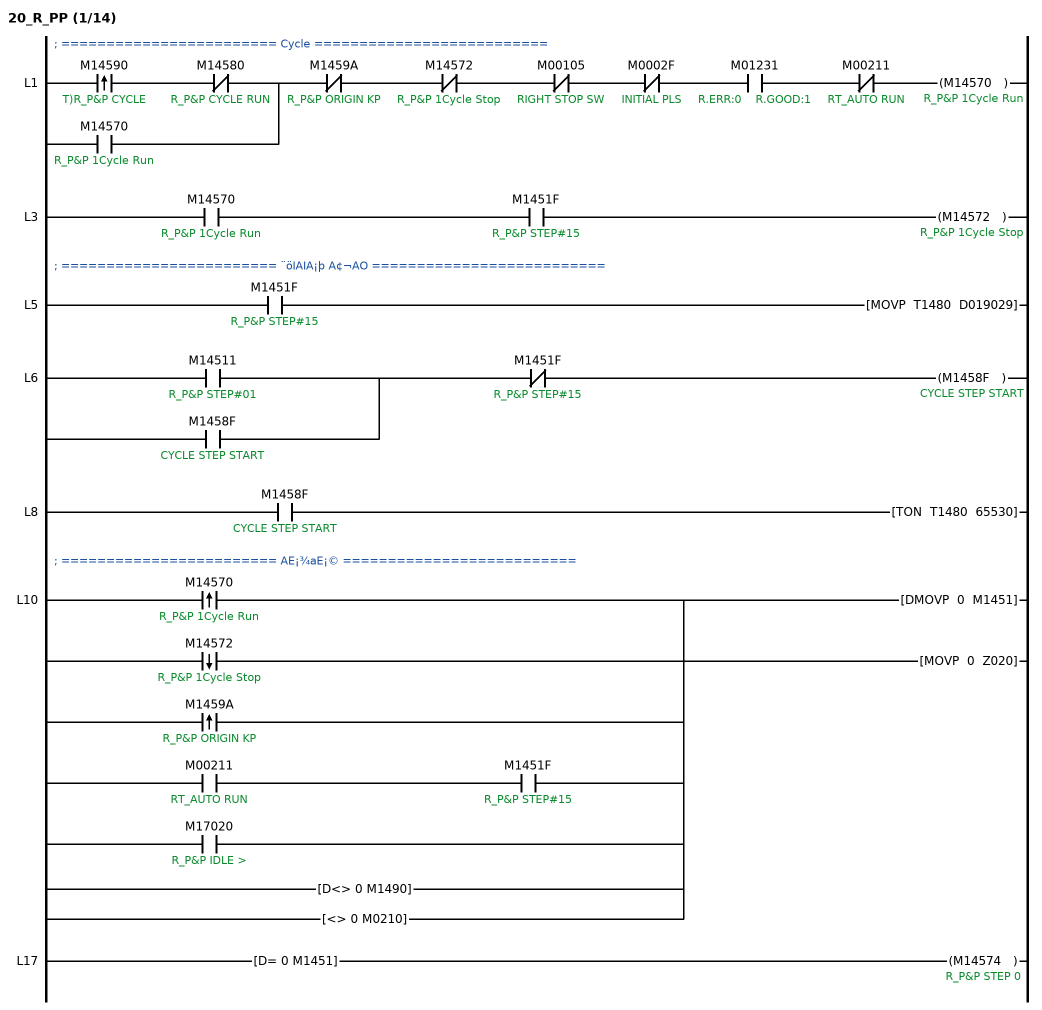
[picture p192: 20_R_PP rungs L1-L17]
// ======================== Cycle ==========================
; L1
LOADP     M14590	// T)R_P&P CYCLE
AND NOT   M14580	// R_P&P CYCLE RUN
OR        M14570	// R_P&P 1Cycle Run
AND NOT   M1459A	// R_P&P ORIGIN KP
AND NOT   M14572	// R_P&P 1Cycle Stop
AND NOT   M00105	// RIGHT STOP SW
AND NOT   M0002F	// INITIAL PLS
AND       M01231	// R.ERR:0    R.GOOD:1
AND NOT   M00211	// RT_AUTO RUN
OUT       M14570	// R_P&P 1Cycle Run
; L3
LOAD      M14570	// R_P&P 1Cycle Run
AND       M1451F	// R_P&P STEP#15
OUT       M14572	// R_P&P 1Cycle Stop
// ======================== ¨öIAIA¡þ A¢¬AO ==========================
; L5
LOAD      M1451F	// R_P&P STEP#15
MOVP      T1480 D019029
; L6
LOAD      M14511	// R_P&P STEP#01
OR        M1458F	// CYCLE STEP START
AND NOT   M1451F	// R_P&P STEP#15
OUT       M1458F	// CYCLE STEP START
; L8
LOAD      M1458F	// CYCLE STEP START
TON       T1480 65530
// ======================== AE¡¾aE¡© ==========================
; L10
LOADP     M14570	// R_P&P 1Cycle Run
ORN       M14572	// R_P&P 1Cycle Stop
ORP       M1459A	// R_P&P ORIGIN KP
LOAD      M00211	// RT_AUTO RUN
AND       M1451F	// R_P&P STEP#15
OR LOAD
OR        M17020	// R_P&P IDLE >
ORD<>     0 M1490
OR<>      0 M0210
DMOVP     0 M1451
MOVP      0 Z020
; L17
LOADD=    0 M1451
OUT       M14574	// R_P&P STEP 0

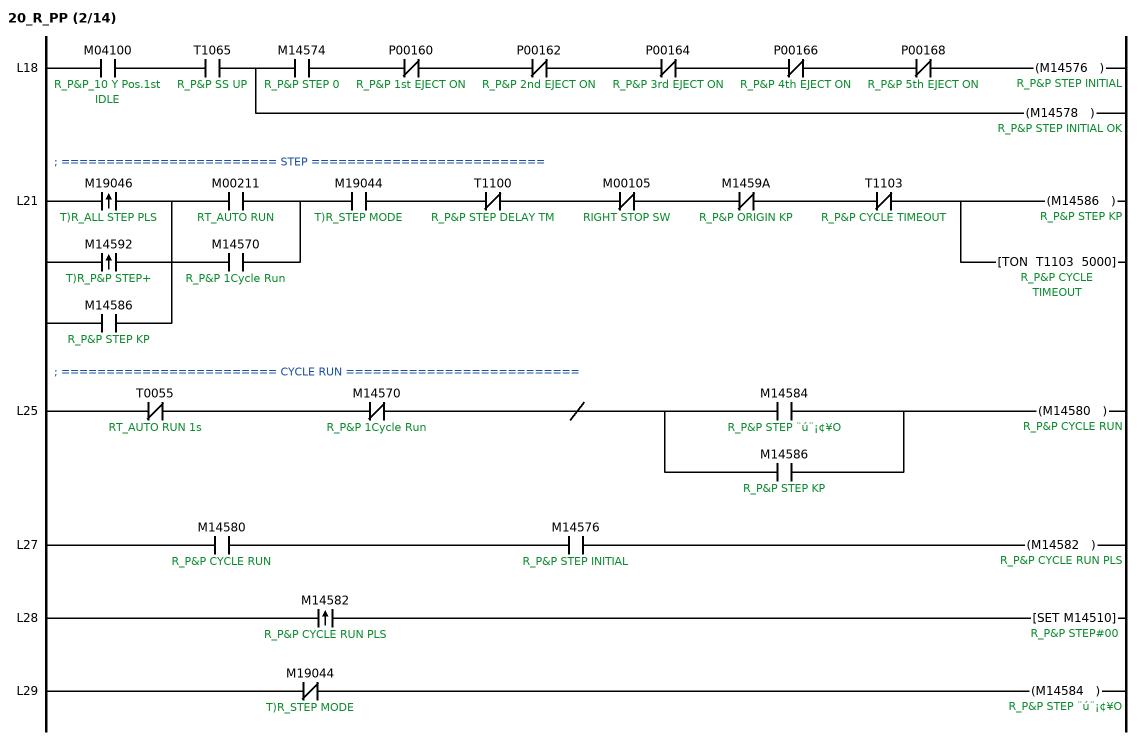
; L18
LOAD      M04100	// R_P&P_10 Y Pos.1st IDLE
AND       T1065	// R_P&P SS UP
MPUSH
AND       M14574	// R_P&P STEP 0
AND NOT   P00160	// R_P&P 1st EJECT ON
AND NOT   P00162	// R_P&P 2nd EJECT ON
AND NOT   P00164	// R_P&P 3rd EJECT ON
AND NOT   P00166	// R_P&P 4th EJECT ON
AND NOT   P00168	// R_P&P 5th EJECT ON
OUT       M14576	// R_P&P STEP INITIAL
MPOP
OUT       M14578	// R_P&P STEP INITIAL OK
// ======================== STEP ==========================
; L21
LOADP     M19046	// T)R_ALL STEP PLS
ORP       M14592	// T)R_P&P STEP+
OR        M14586	// R_P&P STEP KP
LOAD      M00211	// RT_AUTO RUN
OR        M14570	// R_P&P 1Cycle Run
AND LOAD
AND       M19044	// T)R_STEP MODE
AND NOT   T1100	// R_P&P STEP DELAY TM
AND NOT   M00105	// RIGHT STOP SW
AND NOT   M1459A	// R_P&P ORIGIN KP
AND NOT   T1103	// R_P&P CYCLE TIMEOUT
OUT       M14586	// R_P&P STEP KP
TON       T1103 5000	// R_P&P CYCLE TIMEOUT
// ======================== CYCLE RUN ==========================
; L25
LOAD NOT  T0055	// RT_AUTO RUN 1s
AND NOT   M14570	// R_P&P 1Cycle Run
NOT
LOAD      M14584	// R_P&P STEP ¨ú¨¡¢¥O
OR        M14586	// R_P&P STEP KP
AND LOAD
OUT       M14580	// R_P&P CYCLE RUN
; L27
LOAD      M14580	// R_P&P CYCLE RUN
AND       M14576	// R_P&P STEP INITIAL
OUT       M14582	// R_P&P CYCLE RUN PLS
; L28
LOADP     M14582	// R_P&P CYCLE RUN PLS
SET       M14510	// R_P&P STEP#00
; L29
LOAD NOT  M19044	// T)R_STEP MODE
OUT       M14584	// R_P&P STEP ¨ú¨¡¢¥O

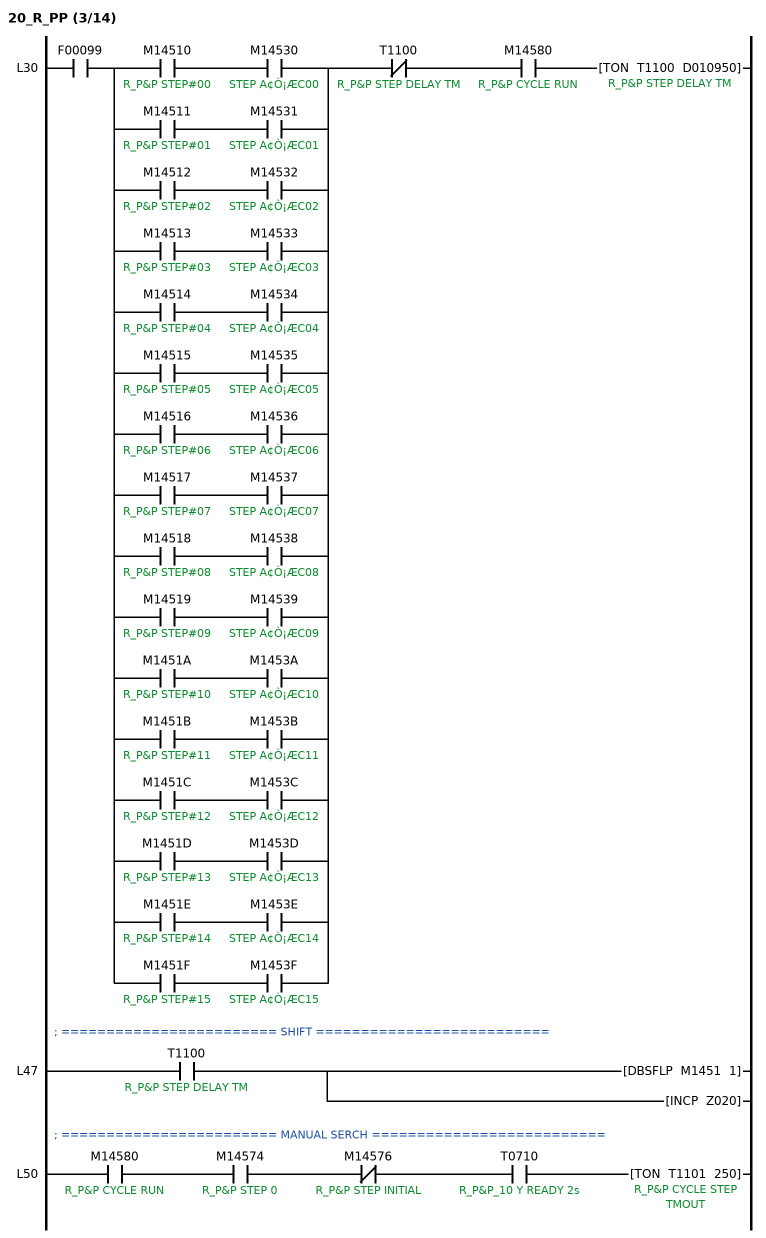
; L30
LOAD      F00099
LOAD      M14510	// R_P&P STEP#00
AND       M14530	// STEP A¢Ò¡ÆC00
LOAD      M14511	// R_P&P STEP#01
AND       M14531	// STEP A¢Ò¡ÆC01
OR LOAD
LOAD      M14512	// R_P&P STEP#02
AND       M14532	// STEP A¢Ò¡ÆC02
OR LOAD
LOAD      M14513	// R_P&P STEP#03
AND       M14533	// STEP A¢Ò¡ÆC03
OR LOAD
LOAD      M14514	// R_P&P STEP#04
AND       M14534	// STEP A¢Ò¡ÆC04
OR LOAD
LOAD      M14515	// R_P&P STEP#05
AND       M14535	// STEP A¢Ò¡ÆC05
OR LOAD
LOAD      M14516	// R_P&P STEP#06
AND       M14536	// STEP A¢Ò¡ÆC06
OR LOAD
LOAD      M14517	// R_P&P STEP#07
AND       M14537	// STEP A¢Ò¡ÆC07
OR LOAD
LOAD      M14518	// R_P&P STEP#08
AND       M14538	// STEP A¢Ò¡ÆC08
OR LOAD
LOAD      M14519	// R_P&P STEP#09
AND       M14539	// STEP A¢Ò¡ÆC09
OR LOAD
LOAD      M1451A	// R_P&P STEP#10
AND       M1453A	// STEP A¢Ò¡ÆC10
OR LOAD
LOAD      M1451B	// R_P&P STEP#11
AND       M1453B	// STEP A¢Ò¡ÆC11
OR LOAD
LOAD      M1451C	// R_P&P STEP#12
AND       M1453C	// STEP A¢Ò¡ÆC12
OR LOAD
LOAD      M1451D	// R_P&P STEP#13
AND       M1453D	// STEP A¢Ò¡ÆC13
OR LOAD
LOAD      M1451E	// R_P&P STEP#14
AND       M1453E	// STEP A¢Ò¡ÆC14
OR LOAD
LOAD      M1451F	// R_P&P STEP#15
AND       M1453F	// STEP A¢Ò¡ÆC15
OR LOAD
AND LOAD
AND NOT   T1100	// R_P&P STEP DELAY TM
AND       M14580	// R_P&P CYCLE RUN
TON       T1100 D010950	// R_P&P STEP DELAY TM
// ======================== SHIFT ==========================
; L47
LOAD      T1100	// R_P&P STEP DELAY TM
DBSFLP    M1451 1
INCP      Z020
// ======================== MANUAL SERCH ==========================
; L50
LOAD      M14580	// R_P&P CYCLE RUN
AND       M14574	// R_P&P STEP 0
AND NOT   M14576	// R_P&P STEP INITIAL
AND       T0710	// R_P&P_10 Y READY 2s
TON       T1101 250	// R_P&P CYCLE STEP TMOUT

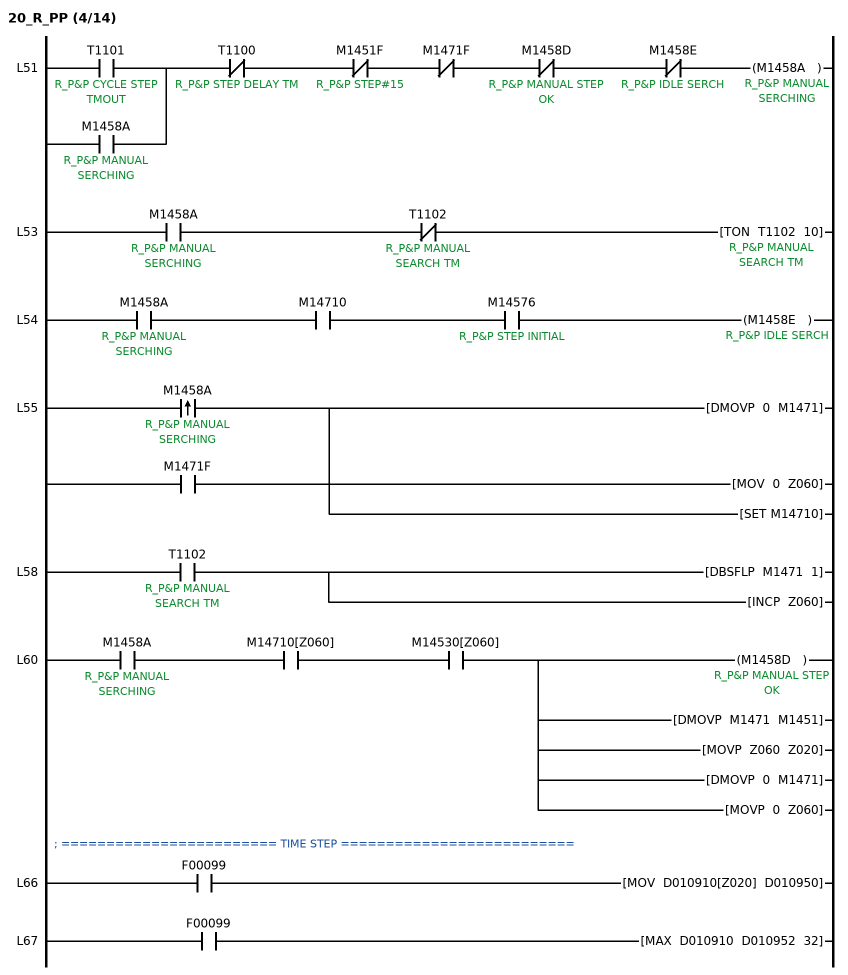
; L51
LOAD      T1101	// R_P&P CYCLE STEP TMOUT
OR        M1458A	// R_P&P MANUAL SERCHING
AND NOT   T1100	// R_P&P STEP DELAY TM
AND NOT   M1451F	// R_P&P STEP#15
AND NOT   M1471F
AND NOT   M1458D	// R_P&P MANUAL STEP OK
AND NOT   M1458E	// R_P&P IDLE SERCH
OUT       M1458A	// R_P&P MANUAL SERCHING
; L53
LOAD      M1458A	// R_P&P MANUAL SERCHING
AND NOT   T1102	// R_P&P MANUAL SEARCH TM
TON       T1102 10	// R_P&P MANUAL SEARCH TM
; L54
LOAD      M1458A	// R_P&P MANUAL SERCHING
AND       M14710
AND       M14576	// R_P&P STEP INITIAL
OUT       M1458E	// R_P&P IDLE SERCH
; L55
LOADP     M1458A	// R_P&P MANUAL SERCHING
OR        M1471F
DMOVP     0 M1471
MOV       0 Z060
SET       M14710
; L58
LOAD      T1102	// R_P&P MANUAL SEARCH TM
DBSFLP    M1471 1
INCP      Z060
; L60
LOAD      M1458A	// R_P&P MANUAL SERCHING
AND       M14710[Z060]
AND       M14530[Z060]
OUT       M1458D	// R_P&P MANUAL STEP OK
DMOVP     M1471 M1451
MOVP      Z060 Z020
DMOVP     0 M1471
MOVP      0 Z060
// ======================== TIME STEP ==========================
; L66
LOAD      F00099
MOV       D010910[Z020] D010950
; L67
LOAD      F00099
MAX       D010910 D010952 32

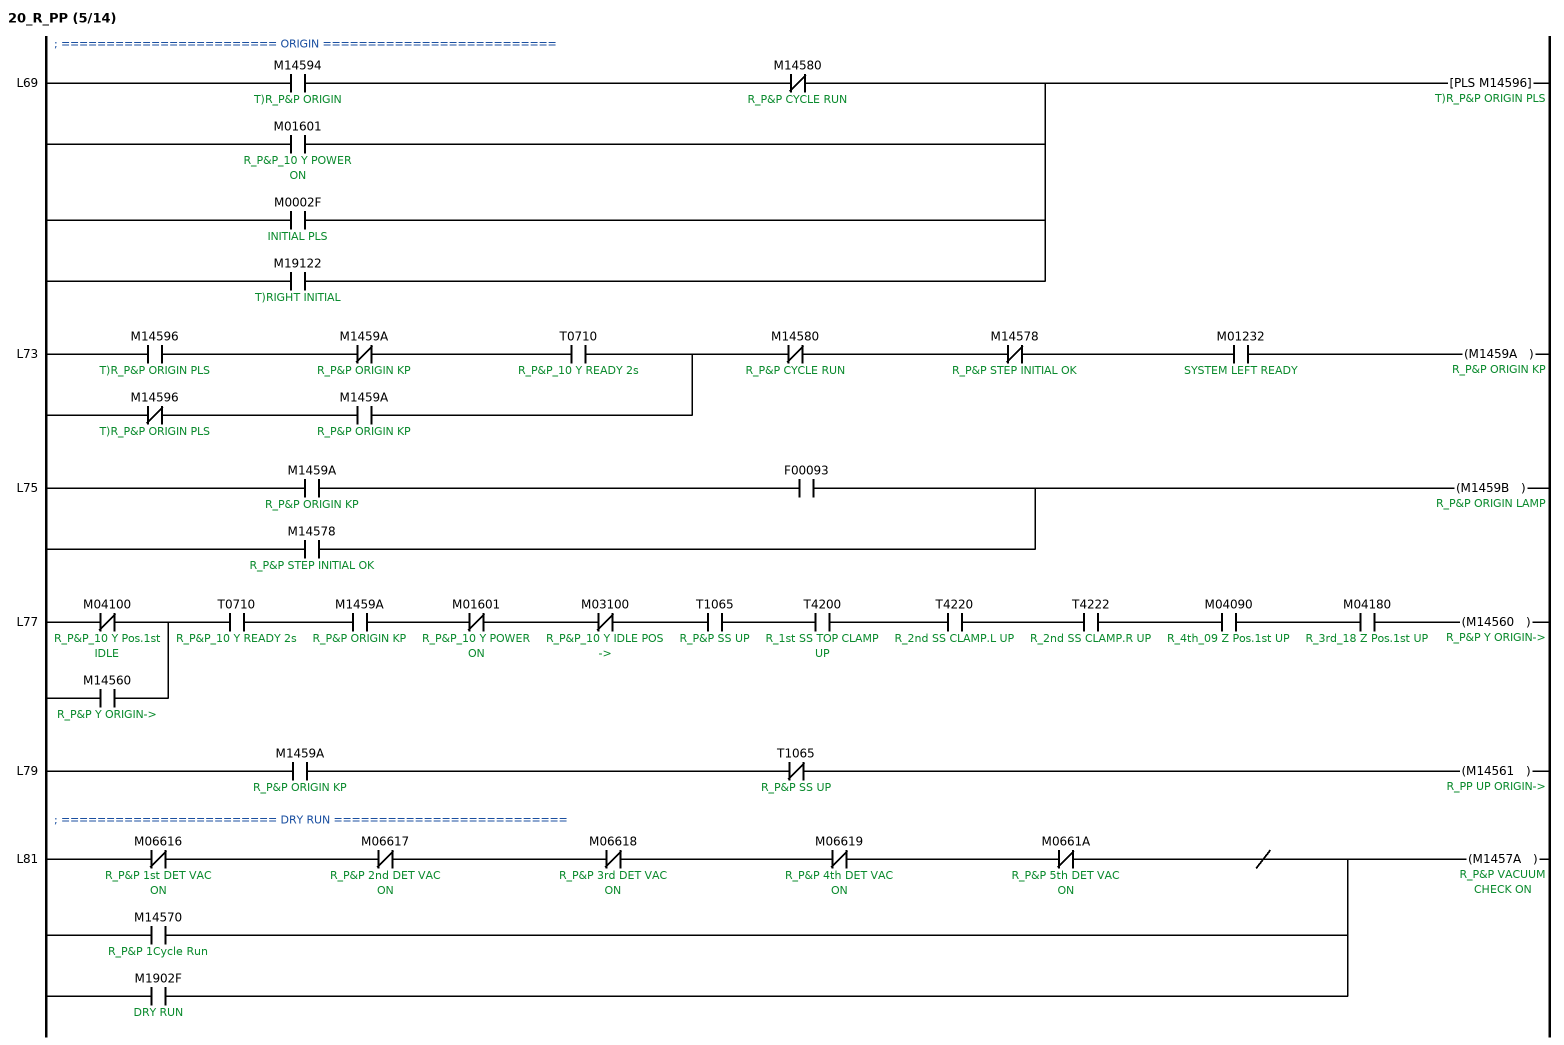
// ======================== ORIGIN ==========================
; L69
LOAD      M14594	// T)R_P&P ORIGIN
AND NOT   M14580	// R_P&P CYCLE RUN
OR        M01601	// R_P&P_10 Y POWER ON
OR        M0002F	// INITIAL PLS
OR        M19122	// T)RIGHT INITIAL
OUTP      M14596	// T)R_P&P ORIGIN PLS
; L73
LOAD      M14596	// T)R_P&P ORIGIN PLS
AND NOT   M1459A	// R_P&P ORIGIN KP
AND       T0710	// R_P&P_10 Y READY 2s
LOAD NOT  M14596	// T)R_P&P ORIGIN PLS
AND       M1459A	// R_P&P ORIGIN KP
OR LOAD
AND NOT   M14580	// R_P&P CYCLE RUN
AND NOT   M14578	// R_P&P STEP INITIAL OK
AND       M01232	// SYSTEM LEFT READY
OUT       M1459A	// R_P&P ORIGIN KP
; L75
LOAD      M1459A	// R_P&P ORIGIN KP
AND       F00093
OR        M14578	// R_P&P STEP INITIAL OK
OUT       M1459B	// R_P&P ORIGIN LAMP
; L77
LOAD NOT  M04100	// R_P&P_10 Y Pos.1st IDLE
OR        M14560	// R_P&P Y ORIGIN->
AND       T0710	// R_P&P_10 Y READY 2s
AND       M1459A	// R_P&P ORIGIN KP
AND NOT   M01601	// R_P&P_10 Y POWER ON
AND NOT   M03100	// R_P&P_10 Y IDLE POS ->
AND       T1065	// R_P&P SS UP
AND       T4200	// R_1st SS TOP CLAMP UP
AND       T4220	// R_2nd SS CLAMP.L UP
AND       T4222	// R_2nd SS CLAMP.R UP
AND       M04090	// R_4th_09 Z Pos.1st UP
AND       M04180	// R_3rd_18 Z Pos.1st UP
OUT       M14560	// R_P&P Y ORIGIN->
; L79
LOAD      M1459A	// R_P&P ORIGIN KP
AND NOT   T1065	// R_P&P SS UP
OUT       M14561	// R_PP UP ORIGIN->
// ======================== DRY RUN ==========================
; L81
LOAD NOT  M06616	// R_P&P 1st DET VAC ON
AND NOT   M06617	// R_P&P 2nd DET VAC ON
AND NOT   M06618	// R_P&P 3rd DET VAC ON
AND NOT   M06619	// R_P&P 4th DET VAC ON
AND NOT   M0661A	// R_P&P 5th DET VAC ON
NOT
OR        M14570	// R_P&P 1Cycle Run
OR        M1902F	// DRY RUN
OUT       M1457A	// R_P&P VACUUM CHECK ON

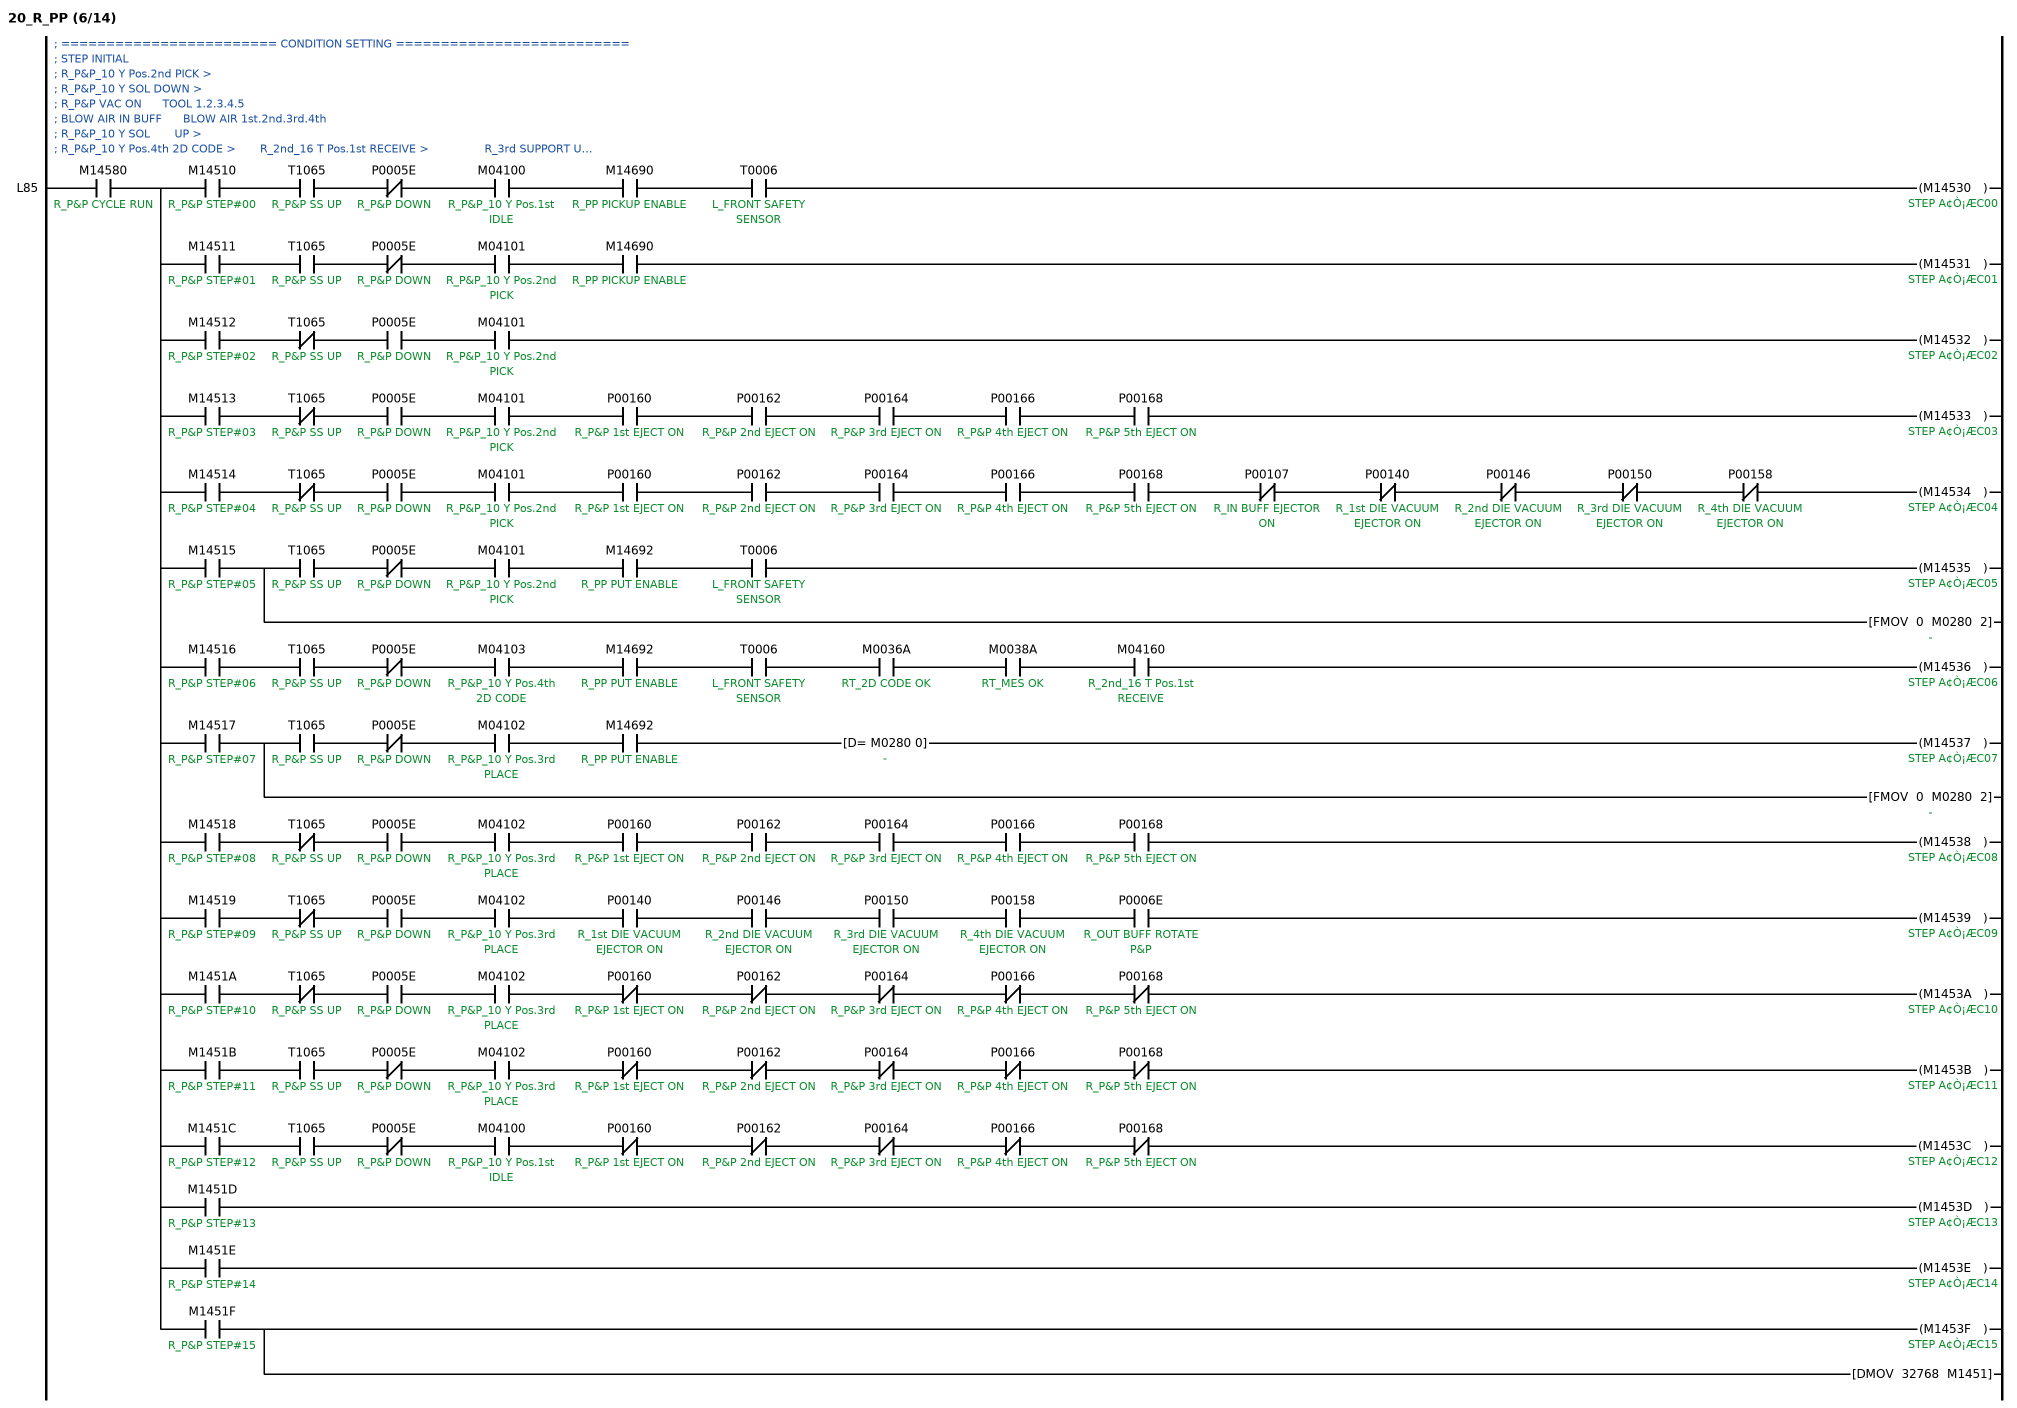
// ======================== CONDITION SETTING ==========================
; L85
LOAD      M14580	// R_P&P CYCLE RUN
MPUSH
AND       M14510	// R_P&P STEP#00
AND       T1065	// R_P&P SS UP
AND NOT   P0005E	// R_P&P DOWN
AND       M04100	// R_P&P_10 Y Pos.1st IDLE
AND       M14690	// R_PP PICKUP ENABLE
AND       T0006	// L_FRONT SAFETY SENSOR
OUT       M14530	// STEP A¢Ò¡ÆC00
MLOAD
AND       M14511	// R_P&P STEP#01
AND       T1065	// R_P&P SS UP
AND NOT   P0005E	// R_P&P DOWN
AND       M04101	// R_P&P_10 Y Pos.2nd PICK
AND       M14690	// R_PP PICKUP ENABLE
OUT       M14531	// STEP A¢Ò¡ÆC01
MLOAD
AND       M14512	// R_P&P STEP#02
AND NOT   T1065	// R_P&P SS UP
AND       P0005E	// R_P&P DOWN
AND       M04101	// R_P&P_10 Y Pos.2nd PICK
OUT       M14532	// STEP A¢Ò¡ÆC02
MLOAD
AND       M14513	// R_P&P STEP#03
AND NOT   T1065	// R_P&P SS UP
AND       P0005E	// R_P&P DOWN
AND       M04101	// R_P&P_10 Y Pos.2nd PICK
AND       P00160	// R_P&P 1st EJECT ON
AND       P00162	// R_P&P 2nd EJECT ON
AND       P00164	// R_P&P 3rd EJECT ON
AND       P00166	// R_P&P 4th EJECT ON
AND       P00168	// R_P&P 5th EJECT ON
OUT       M14533	// STEP A¢Ò¡ÆC03
MLOAD
AND       M14514	// R_P&P STEP#04
AND NOT   T1065	// R_P&P SS UP
AND       P0005E	// R_P&P DOWN
AND       M04101	// R_P&P_10 Y Pos.2nd PICK
AND       P00160	// R_P&P 1st EJECT ON
AND       P00162	// R_P&P 2nd EJECT ON
AND       P00164	// R_P&P 3rd EJECT ON
AND       P00166	// R_P&P 4th EJECT ON
AND       P00168	// R_P&P 5th EJECT ON
AND NOT   P00107	// R_IN BUFF EJECTOR ON
AND NOT   P00140	// R_1st DIE VACUUM EJECTOR ON
AND NOT   P00146	// R_2nd DIE VACUUM EJECTOR ON
AND NOT   P00150	// R_3rd DIE VACUUM EJECTOR ON
AND NOT   P00158	// R_4th DIE VACUUM EJECTOR ON
OUT       M14534	// STEP A¢Ò¡ÆC04
MLOAD
AND       M14515	// R_P&P STEP#05
MPUSH
AND       T1065	// R_P&P SS UP
AND NOT   P0005E	// R_P&P DOWN
AND       M04101	// R_P&P_10 Y Pos.2nd PICK
AND       M14692	// R_PP PUT ENABLE
AND       T0006	// L_FRONT SAFETY SENSOR
OUT       M14535	// STEP A¢Ò¡ÆC05
MPOP
FMOV      0 M0280 2	// -
MLOAD
AND       M14516	// R_P&P STEP#06
AND       T1065	// R_P&P SS UP
AND NOT   P0005E	// R_P&P DOWN
AND       M04103	// R_P&P_10 Y Pos.4th 2D CODE
AND       M14692	// R_PP PUT ENABLE
AND       T0006	// L_FRONT SAFETY SENSOR
AND       M0036A	// RT_2D CODE OK
AND       M0038A	// RT_MES OK
AND       M04160	// R_2nd_16 T Pos.1st RECEIVE
OUT       M14536	// STEP A¢Ò¡ÆC06
MLOAD
AND       M14517	// R_P&P STEP#07
MPUSH
AND       T1065	// R_P&P SS UP
AND NOT   P0005E	// R_P&P DOWN
AND       M04102	// R_P&P_10 Y Pos.3rd PLACE
AND       M14692	// R_PP PUT ENABLE
ANDD=     M0280 0	// -
OUT       M14537	// STEP A¢Ò¡ÆC07
MPOP
FMOV      0 M0280 2	// -
MLOAD
AND       M14518	// R_P&P STEP#08
AND NOT   T1065	// R_P&P SS UP
AND       P0005E	// R_P&P DOWN
AND       M04102	// R_P&P_10 Y Pos.3rd PLACE
AND       P00160	// R_P&P 1st EJECT ON
AND       P00162	// R_P&P 2nd EJECT ON
AND       P00164	// R_P&P 3rd EJECT ON
AND       P00166	// R_P&P 4th EJECT ON
AND       P00168	// R_P&P 5th EJECT ON
OUT       M14538	// STEP A¢Ò¡ÆC08
MLOAD
AND       M14519	// R_P&P STEP#09
AND NOT   T1065	// R_P&P SS UP
AND       P0005E	// R_P&P DOWN
AND       M04102	// R_P&P_10 Y Pos.3rd PLACE
AND       P00140	// R_1st DIE VACUUM EJECTOR ON
AND       P00146	// R_2nd DIE VACUUM EJECTOR ON
AND       P00150	// R_3rd DIE VACUUM EJECTOR ON
AND       P00158	// R_4th DIE VACUUM EJECTOR ON
AND       P0006E	// R_OUT BUFF ROTATE      P&P
OUT       M14539	// STEP A¢Ò¡ÆC09
MLOAD
AND       M1451A	// R_P&P STEP#10
AND NOT   T1065	// R_P&P SS UP
AND       P0005E	// R_P&P DOWN
AND       M04102	// R_P&P_10 Y Pos.3rd PLACE
AND NOT   P00160	// R_P&P 1st EJECT ON
AND NOT   P00162	// R_P&P 2nd EJECT ON
AND NOT   P00164	// R_P&P 3rd EJECT ON
AND NOT   P00166	// R_P&P 4th EJECT ON
AND NOT   P00168	// R_P&P 5th EJECT ON
OUT       M1453A	// STEP A¢Ò¡ÆC10
MLOAD
AND       M1451B	// R_P&P STEP#11
AND       T1065	// R_P&P SS UP
AND NOT   P0005E	// R_P&P DOWN
AND       M04102	// R_P&P_10 Y Pos.3rd PLACE
AND NOT   P00160	// R_P&P 1st EJECT ON
AND NOT   P00162	// R_P&P 2nd EJECT ON
AND NOT   P00164	// R_P&P 3rd EJECT ON
AND NOT   P00166	// R_P&P 4th EJECT ON
AND NOT   P00168	// R_P&P 5th EJECT ON
OUT       M1453B	// STEP A¢Ò¡ÆC11
MLOAD
AND       M1451C	// R_P&P STEP#12
AND       T1065	// R_P&P SS UP
AND NOT   P0005E	// R_P&P DOWN
AND       M04100	// R_P&P_10 Y Pos.1st IDLE
AND NOT   P00160	// R_P&P 1st EJECT ON
AND NOT   P00162	// R_P&P 2nd EJECT ON
AND NOT   P00164	// R_P&P 3rd EJECT ON
AND NOT   P00166	// R_P&P 4th EJECT ON
AND NOT   P00168	// R_P&P 5th EJECT ON
OUT       M1453C	// STEP A¢Ò¡ÆC12
MLOAD
AND       M1451D	// R_P&P STEP#13
OUT       M1453D	// STEP A¢Ò¡ÆC13
MLOAD
AND       M1451E	// R_P&P STEP#14
OUT       M1453E	// STEP A¢Ò¡ÆC14
MPOP
AND       M1451F	// R_P&P STEP#15
OUT       M1453F	// STEP A¢Ò¡ÆC15
DMOV      32768 M1451
// output comment: STEP INITIAL
// output comment: R_P&P_10 Y Pos.2nd PICK >
// output comment: R_P&P_10 Y SOL DOWN >
// output comment: R_P&P VAC ON      TOOL 1.2.3.4.5
// output comment: BLOW AIR IN BUFF      BLOW AIR 1st.2nd.3rd.4th
// output comment: R_P&P_10 Y SOL       UP >
// output comment: R_P&P_10 Y Pos.4th 2D CODE >       R_2nd_16 T Pos.1st RECEIVE >                R_3rd SUPPORT UP
// output comment: R_P&P_10 Y Pos.3rd PLACE >
// output comment: R_P&P_10 Y SOL       DOWN >
// output comment: R_P&P BLOW AIR      TOOL 1.2.3.4.5
// output comment: R_P&P_10 Y SOL       UP >
// output comment: R_P&P_10 Y Pos.1st IDLE >

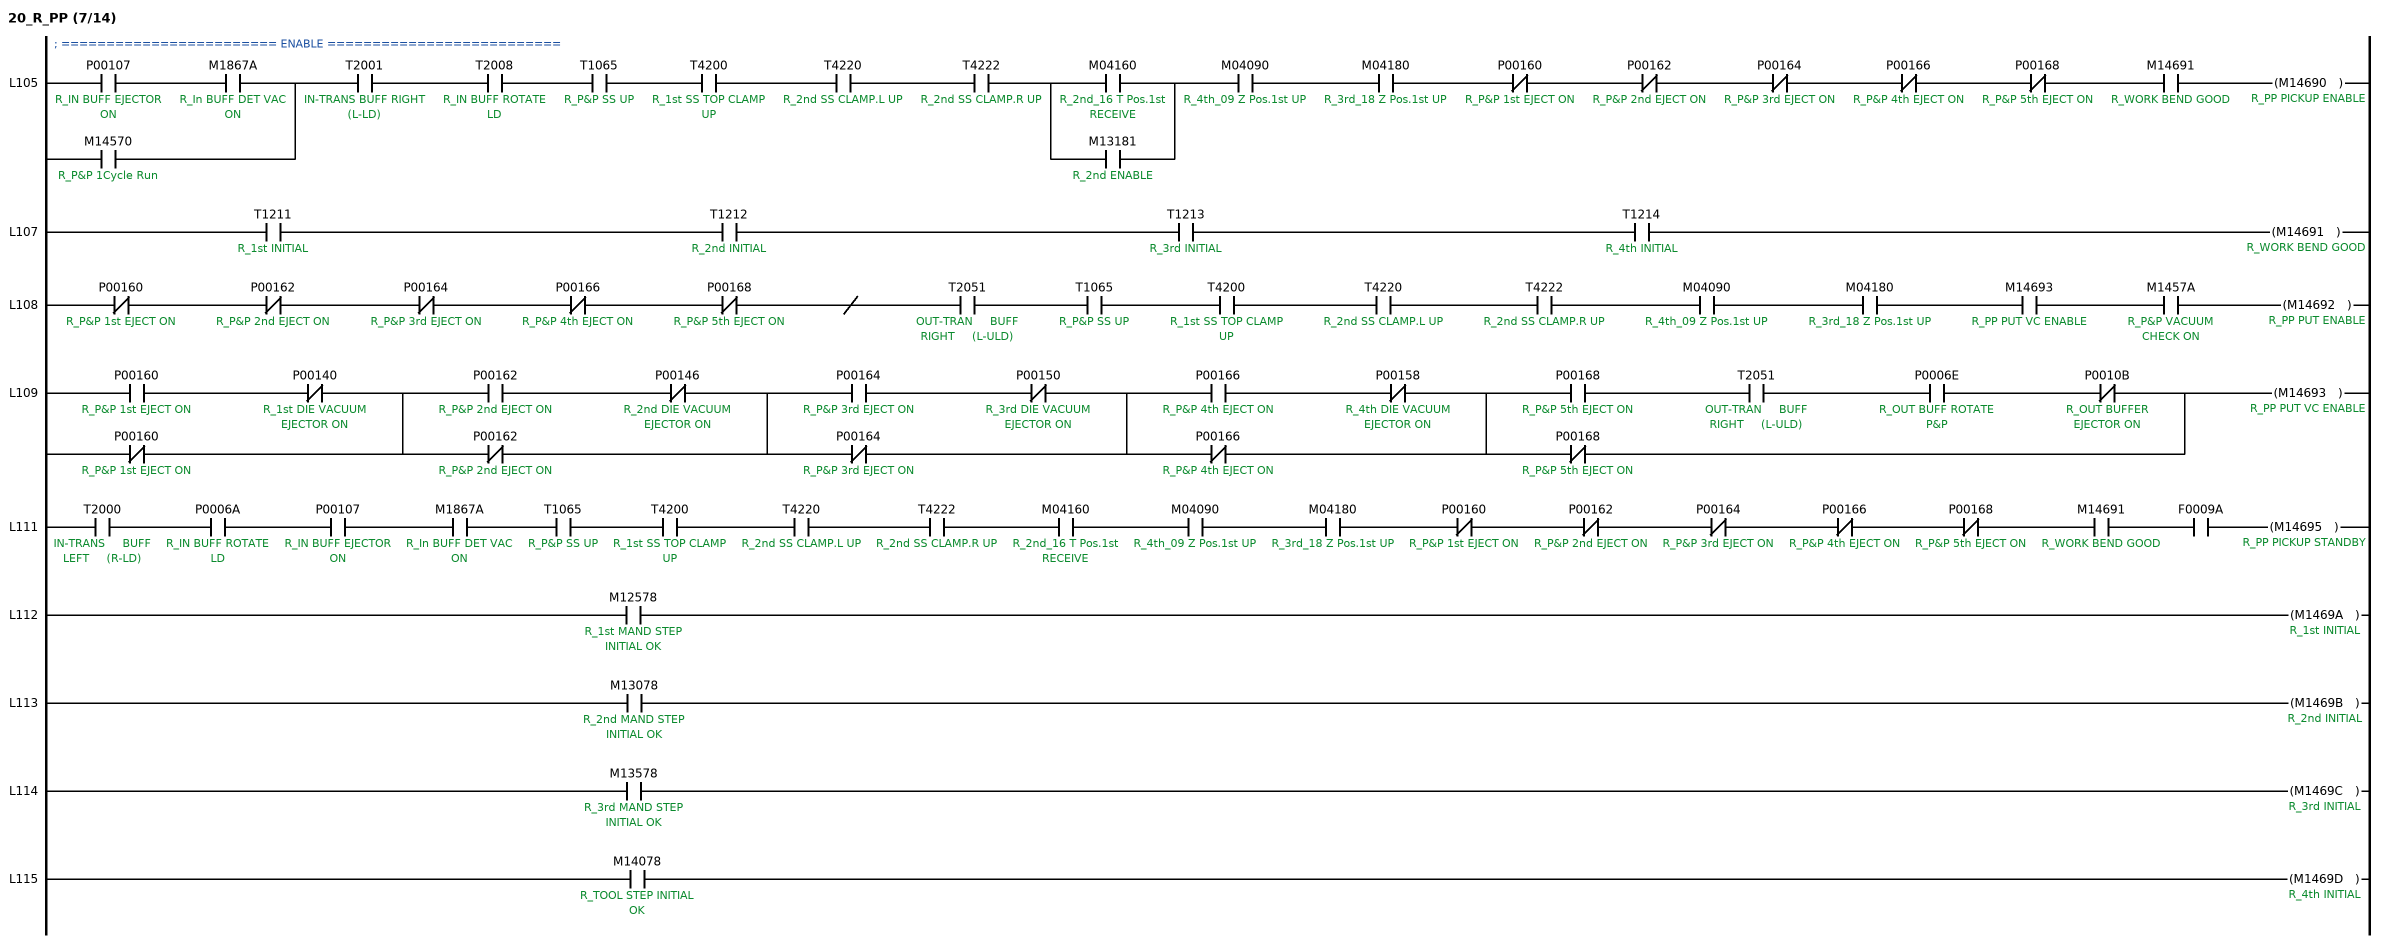
// ======================== ENABLE ==========================
; L105
LOAD      P00107	// R_IN BUFF EJECTOR ON
AND       M1867A	// R_In BUFF DET VAC ON
OR        M14570	// R_P&P 1Cycle Run
AND       T2001	// IN-TRANS BUFF RIGHT     (L-LD)
AND       T2008	// R_IN BUFF ROTATE      LD
AND       T1065	// R_P&P SS UP
AND       T4200	// R_1st SS TOP CLAMP UP
AND       T4220	// R_2nd SS CLAMP.L UP
AND       T4222	// R_2nd SS CLAMP.R UP
LOAD      M04160	// R_2nd_16 T Pos.1st RECEIVE
OR        M13181	// R_2nd ENABLE
AND LOAD
AND       M04090	// R_4th_09 Z Pos.1st UP
AND       M04180	// R_3rd_18 Z Pos.1st UP
AND NOT   P00160	// R_P&P 1st EJECT ON
AND NOT   P00162	// R_P&P 2nd EJECT ON
AND NOT   P00164	// R_P&P 3rd EJECT ON
AND NOT   P00166	// R_P&P 4th EJECT ON
AND NOT   P00168	// R_P&P 5th EJECT ON
AND       M14691	// R_WORK BEND GOOD
OUT       M14690	// R_PP PICKUP ENABLE
; L107
LOAD      T1211	// R_1st INITIAL
AND       T1212	// R_2nd INITIAL
AND       T1213	// R_3rd INITIAL
AND       T1214	// R_4th INITIAL
OUT       M14691	// R_WORK BEND GOOD
; L108
LOAD NOT  P00160	// R_P&P 1st EJECT ON
AND NOT   P00162	// R_P&P 2nd EJECT ON
AND NOT   P00164	// R_P&P 3rd EJECT ON
AND NOT   P00166	// R_P&P 4th EJECT ON
AND NOT   P00168	// R_P&P 5th EJECT ON
NOT
AND       T2051	// OUT-TRAN     BUFF     RIGHT     (L-ULD)
AND       T1065	// R_P&P SS UP
AND       T4200	// R_1st SS TOP CLAMP UP
AND       T4220	// R_2nd SS CLAMP.L UP
AND       T4222	// R_2nd SS CLAMP.R UP
AND       M04090	// R_4th_09 Z Pos.1st UP
AND       M04180	// R_3rd_18 Z Pos.1st UP
AND       M14693	// R_PP PUT VC ENABLE
AND       M1457A	// R_P&P VACUUM CHECK ON
OUT       M14692	// R_PP PUT ENABLE
; L109
LOAD      P00160	// R_P&P 1st EJECT ON
AND NOT   P00140	// R_1st DIE VACUUM EJECTOR ON
OR NOT    P00160	// R_P&P 1st EJECT ON
LOAD      P00162	// R_P&P 2nd EJECT ON
AND NOT   P00146	// R_2nd DIE VACUUM EJECTOR ON
OR NOT    P00162	// R_P&P 2nd EJECT ON
AND LOAD
LOAD      P00164	// R_P&P 3rd EJECT ON
AND NOT   P00150	// R_3rd DIE VACUUM EJECTOR ON
OR NOT    P00164	// R_P&P 3rd EJECT ON
AND LOAD
LOAD      P00166	// R_P&P 4th EJECT ON
AND NOT   P00158	// R_4th DIE VACUUM EJECTOR ON
OR NOT    P00166	// R_P&P 4th EJECT ON
AND LOAD
LOAD      P00168	// R_P&P 5th EJECT ON
AND       T2051	// OUT-TRAN     BUFF     RIGHT     (L-ULD)
AND       P0006E	// R_OUT BUFF ROTATE      P&P
AND NOT   P0010B	// R_OUT BUFFER EJECTOR ON
OR NOT    P00168	// R_P&P 5th EJECT ON
AND LOAD
OUT       M14693	// R_PP PUT VC ENABLE
; L111
LOAD      T2000	// IN-TRANS     BUFF     LEFT     (R-LD)
AND       P0006A	// R_IN BUFF ROTATE      LD
AND       P00107	// R_IN BUFF EJECTOR ON
AND       M1867A	// R_In BUFF DET VAC ON
AND       T1065	// R_P&P SS UP
AND       T4200	// R_1st SS TOP CLAMP UP
AND       T4220	// R_2nd SS CLAMP.L UP
AND       T4222	// R_2nd SS CLAMP.R UP
AND       M04160	// R_2nd_16 T Pos.1st RECEIVE
AND       M04090	// R_4th_09 Z Pos.1st UP
AND       M04180	// R_3rd_18 Z Pos.1st UP
AND NOT   P00160	// R_P&P 1st EJECT ON
AND NOT   P00162	// R_P&P 2nd EJECT ON
AND NOT   P00164	// R_P&P 3rd EJECT ON
AND NOT   P00166	// R_P&P 4th EJECT ON
AND NOT   P00168	// R_P&P 5th EJECT ON
AND       M14691	// R_WORK BEND GOOD
AND       F0009A
OUT       M14695	// R_PP PICKUP STANDBY
; L112
LOAD      M12578	// R_1st MAND STEP INITIAL OK
OUT       M1469A	// R_1st INITIAL
; L113
LOAD      M13078	// R_2nd MAND STEP INITIAL OK
OUT       M1469B	// R_2nd INITIAL
; L114
LOAD      M13578	// R_3rd MAND STEP INITIAL OK
OUT       M1469C	// R_3rd INITIAL
; L115
LOAD      M14078	// R_TOOL STEP INITIAL OK
OUT       M1469D	// R_4th INITIAL

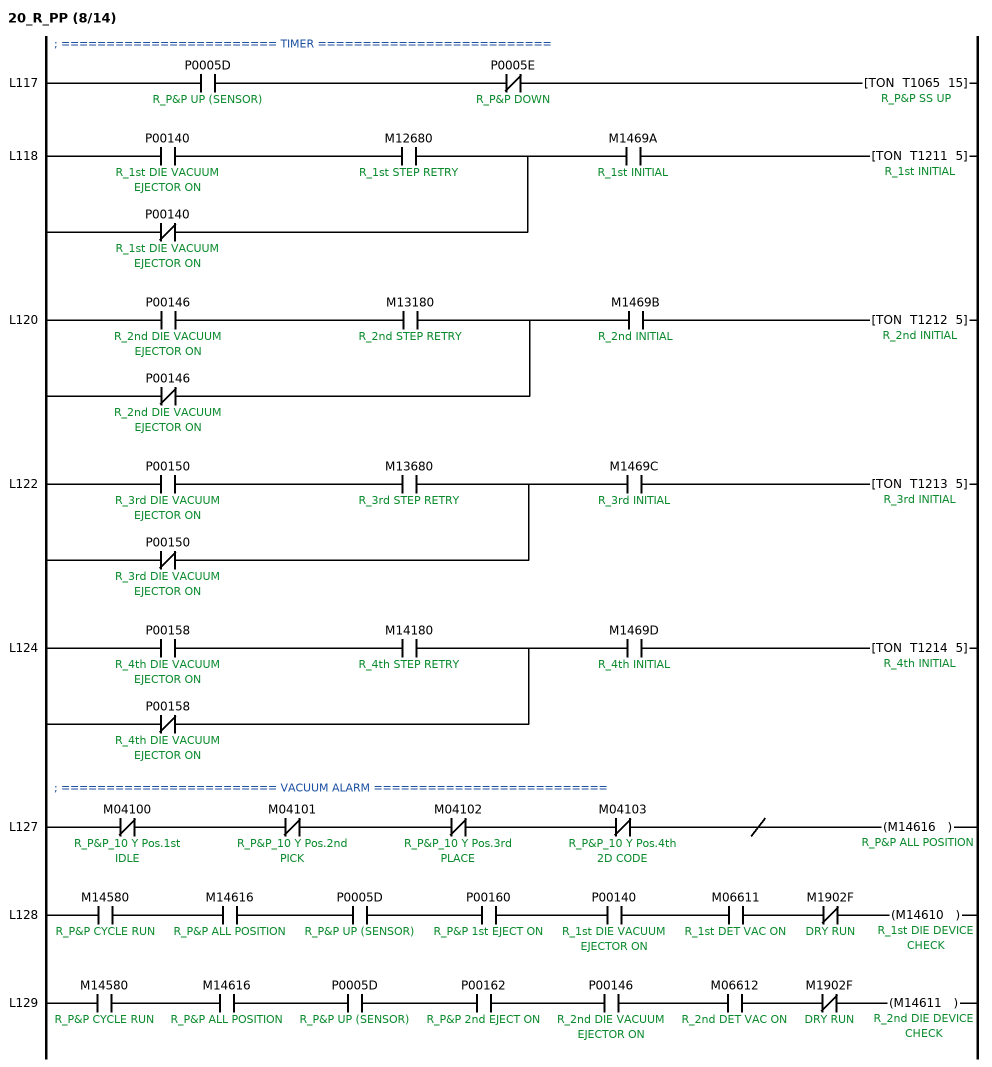
// ======================== TIMER ==========================
; L117
LOAD      P0005D	// R_P&P UP (SENSOR)
AND NOT   P0005E	// R_P&P DOWN
TON       T1065 15	// R_P&P SS UP
; L118
LOAD      P00140	// R_1st DIE VACUUM EJECTOR ON
AND       M12680	// R_1st STEP RETRY
OR NOT    P00140	// R_1st DIE VACUUM EJECTOR ON
AND       M1469A	// R_1st INITIAL
TON       T1211 5	// R_1st INITIAL
; L120
LOAD      P00146	// R_2nd DIE VACUUM EJECTOR ON
AND       M13180	// R_2nd STEP RETRY
OR NOT    P00146	// R_2nd DIE VACUUM EJECTOR ON
AND       M1469B	// R_2nd INITIAL
TON       T1212 5	// R_2nd INITIAL
; L122
LOAD      P00150	// R_3rd DIE VACUUM EJECTOR ON
AND       M13680	// R_3rd STEP RETRY
OR NOT    P00150	// R_3rd DIE VACUUM EJECTOR ON
AND       M1469C	// R_3rd INITIAL
TON       T1213 5	// R_3rd INITIAL
; L124
LOAD      P00158	// R_4th DIE VACUUM EJECTOR ON
AND       M14180	// R_4th STEP RETRY
OR NOT    P00158	// R_4th DIE VACUUM EJECTOR ON
AND       M1469D	// R_4th INITIAL
TON       T1214 5	// R_4th INITIAL
// ======================== VACUUM ALARM ==========================
; L127
LOAD NOT  M04100	// R_P&P_10 Y Pos.1st IDLE
AND NOT   M04101	// R_P&P_10 Y Pos.2nd PICK
AND NOT   M04102	// R_P&P_10 Y Pos.3rd PLACE
AND NOT   M04103	// R_P&P_10 Y Pos.4th 2D CODE
NOT
OUT       M14616	// R_P&P ALL POSITION
; L128
LOAD      M14580	// R_P&P CYCLE RUN
AND       M14616	// R_P&P ALL POSITION
AND       P0005D	// R_P&P UP (SENSOR)
AND       P00160	// R_P&P 1st EJECT ON
AND       P00140	// R_1st DIE VACUUM EJECTOR ON
AND       M06611	// R_1st DET VAC ON
AND NOT   M1902F	// DRY RUN
OUT       M14610	// R_1st DIE DEVICE CHECK
; L129
LOAD      M14580	// R_P&P CYCLE RUN
AND       M14616	// R_P&P ALL POSITION
AND       P0005D	// R_P&P UP (SENSOR)
AND       P00162	// R_P&P 2nd EJECT ON
AND       P00146	// R_2nd DIE VACUUM EJECTOR ON
AND       M06612	// R_2nd DET VAC ON
AND NOT   M1902F	// DRY RUN
OUT       M14611	// R_2nd DIE DEVICE CHECK

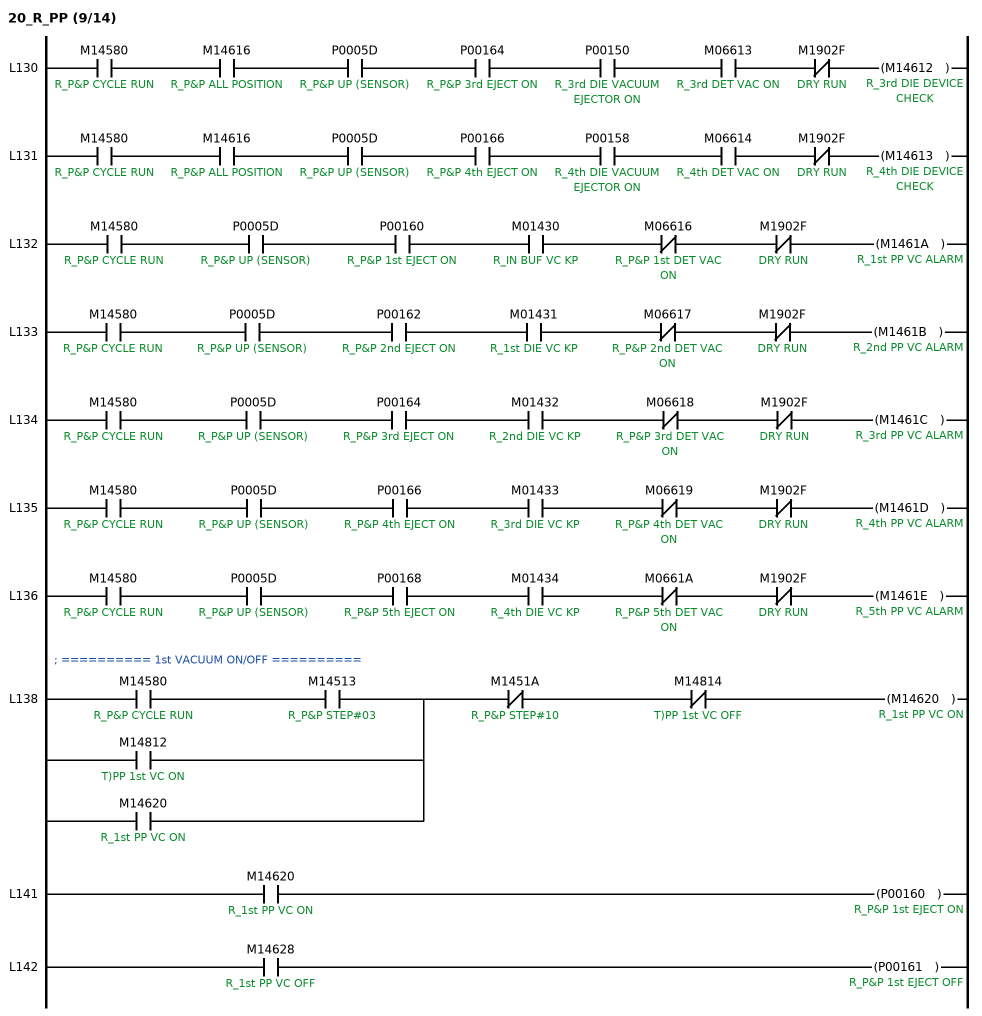
; L130
LOAD      M14580	// R_P&P CYCLE RUN
AND       M14616	// R_P&P ALL POSITION
AND       P0005D	// R_P&P UP (SENSOR)
AND       P00164	// R_P&P 3rd EJECT ON
AND       P00150	// R_3rd DIE VACUUM EJECTOR ON
AND       M06613	// R_3rd DET VAC ON
AND NOT   M1902F	// DRY RUN
OUT       M14612	// R_3rd DIE DEVICE CHECK
; L131
LOAD      M14580	// R_P&P CYCLE RUN
AND       M14616	// R_P&P ALL POSITION
AND       P0005D	// R_P&P UP (SENSOR)
AND       P00166	// R_P&P 4th EJECT ON
AND       P00158	// R_4th DIE VACUUM EJECTOR ON
AND       M06614	// R_4th DET VAC ON
AND NOT   M1902F	// DRY RUN
OUT       M14613	// R_4th DIE DEVICE CHECK
; L132
LOAD      M14580	// R_P&P CYCLE RUN
AND       P0005D	// R_P&P UP (SENSOR)
AND       P00160	// R_P&P 1st EJECT ON
AND       M01430	// R_IN BUF VC KP
AND NOT   M06616	// R_P&P 1st DET VAC ON
AND NOT   M1902F	// DRY RUN
OUT       M1461A	// R_1st PP VC ALARM
; L133
LOAD      M14580	// R_P&P CYCLE RUN
AND       P0005D	// R_P&P UP (SENSOR)
AND       P00162	// R_P&P 2nd EJECT ON
AND       M01431	// R_1st DIE VC KP
AND NOT   M06617	// R_P&P 2nd DET VAC ON
AND NOT   M1902F	// DRY RUN
OUT       M1461B	// R_2nd PP VC ALARM
; L134
LOAD      M14580	// R_P&P CYCLE RUN
AND       P0005D	// R_P&P UP (SENSOR)
AND       P00164	// R_P&P 3rd EJECT ON
AND       M01432	// R_2nd DIE VC KP
AND NOT   M06618	// R_P&P 3rd DET VAC ON
AND NOT   M1902F	// DRY RUN
OUT       M1461C	// R_3rd PP VC ALARM
; L135
LOAD      M14580	// R_P&P CYCLE RUN
AND       P0005D	// R_P&P UP (SENSOR)
AND       P00166	// R_P&P 4th EJECT ON
AND       M01433	// R_3rd DIE VC KP
AND NOT   M06619	// R_P&P 4th DET VAC ON
AND NOT   M1902F	// DRY RUN
OUT       M1461D	// R_4th PP VC ALARM
; L136
LOAD      M14580	// R_P&P CYCLE RUN
AND       P0005D	// R_P&P UP (SENSOR)
AND       P00168	// R_P&P 5th EJECT ON
AND       M01434	// R_4th DIE VC KP
AND NOT   M0661A	// R_P&P 5th DET VAC ON
AND NOT   M1902F	// DRY RUN
OUT       M1461E	// R_5th PP VC ALARM
// ========== 1st VACUUM ON/OFF ==========
; L138
LOAD      M14580	// R_P&P CYCLE RUN
AND       M14513	// R_P&P STEP#03
OR        M14812	// T)PP 1st VC ON
OR        M14620	// R_1st PP VC ON
AND NOT   M1451A	// R_P&P STEP#10
AND NOT   M14814	// T)PP 1st VC OFF
OUT       M14620	// R_1st PP VC ON
; L141
LOAD      M14620	// R_1st PP VC ON
OUT       P00160	// R_P&P 1st EJECT ON
; L142
LOAD      M14628	// R_1st PP VC OFF
OUT       P00161	// R_P&P 1st EJECT OFF

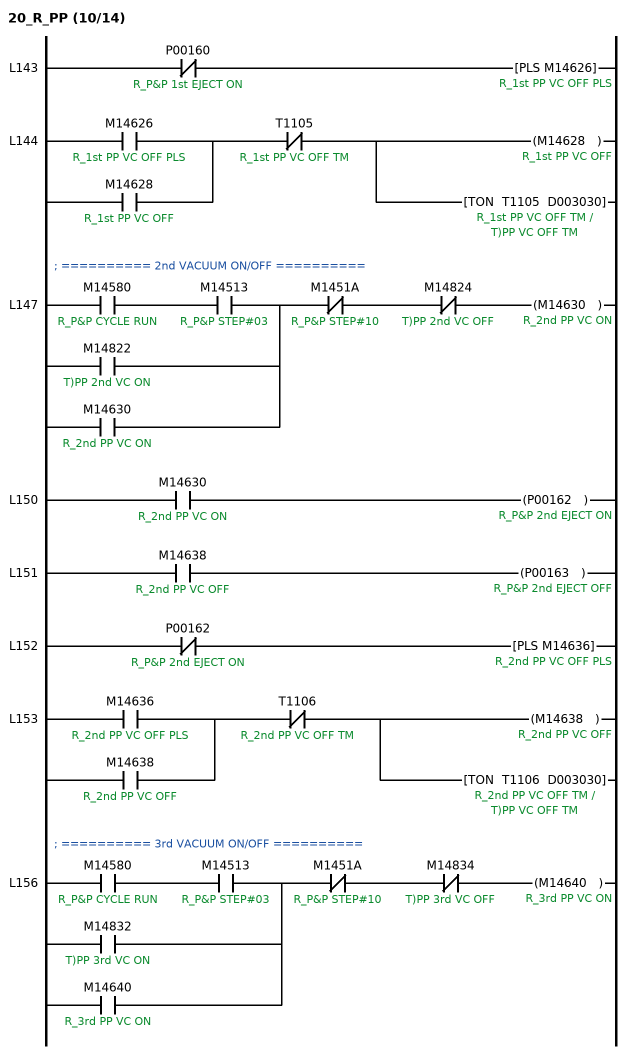
; L143
LOAD NOT  P00160	// R_P&P 1st EJECT ON
OUTP      M14626	// R_1st PP VC OFF PLS
; L144
LOAD      M14626	// R_1st PP VC OFF PLS
OR        M14628	// R_1st PP VC OFF
AND NOT   T1105	// R_1st PP VC OFF TM
OUT       M14628	// R_1st PP VC OFF
TON       T1105 D003030	// R_1st PP VC OFF TM / T)PP VC OFF TM
// ========== 2nd VACUUM ON/OFF ==========
; L147
LOAD      M14580	// R_P&P CYCLE RUN
AND       M14513	// R_P&P STEP#03
OR        M14822	// T)PP 2nd VC ON
OR        M14630	// R_2nd PP VC ON
AND NOT   M1451A	// R_P&P STEP#10
AND NOT   M14824	// T)PP 2nd VC OFF
OUT       M14630	// R_2nd PP VC ON
; L150
LOAD      M14630	// R_2nd PP VC ON
OUT       P00162	// R_P&P 2nd EJECT ON
; L151
LOAD      M14638	// R_2nd PP VC OFF
OUT       P00163	// R_P&P 2nd EJECT OFF
; L152
LOAD NOT  P00162	// R_P&P 2nd EJECT ON
OUTP      M14636	// R_2nd PP VC OFF PLS
; L153
LOAD      M14636	// R_2nd PP VC OFF PLS
OR        M14638	// R_2nd PP VC OFF
AND NOT   T1106	// R_2nd PP VC OFF TM
OUT       M14638	// R_2nd PP VC OFF
TON       T1106 D003030	// R_2nd PP VC OFF TM / T)PP VC OFF TM
// ========== 3rd VACUUM ON/OFF ==========
; L156
LOAD      M14580	// R_P&P CYCLE RUN
AND       M14513	// R_P&P STEP#03
OR        M14832	// T)PP 3rd VC ON
OR        M14640	// R_3rd PP VC ON
AND NOT   M1451A	// R_P&P STEP#10
AND NOT   M14834	// T)PP 3rd VC OFF
OUT       M14640	// R_3rd PP VC ON

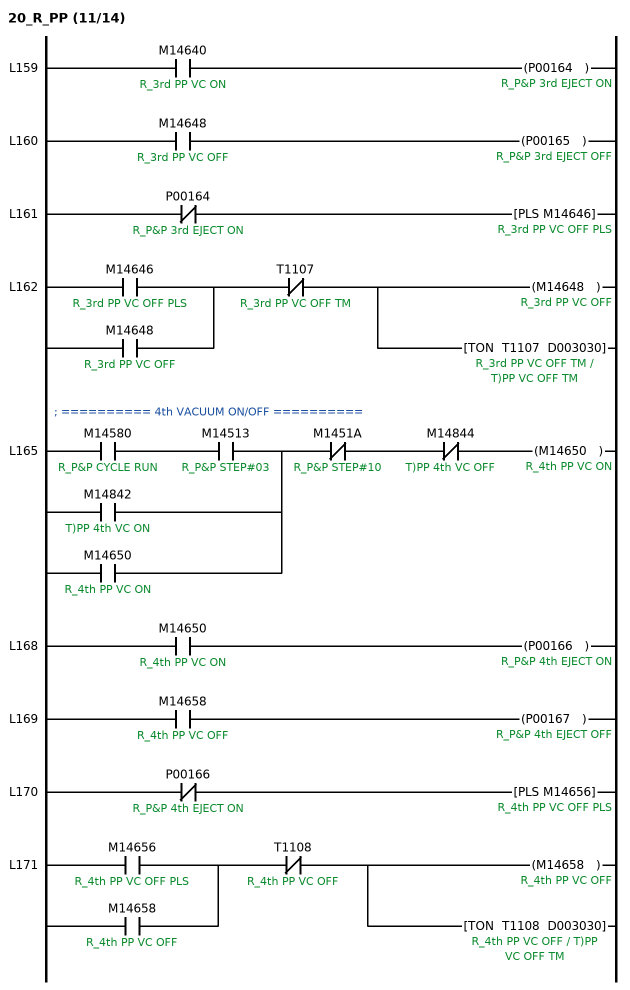
; L159
LOAD      M14640	// R_3rd PP VC ON
OUT       P00164	// R_P&P 3rd EJECT ON
; L160
LOAD      M14648	// R_3rd PP VC OFF
OUT       P00165	// R_P&P 3rd EJECT OFF
; L161
LOAD NOT  P00164	// R_P&P 3rd EJECT ON
OUTP      M14646	// R_3rd PP VC OFF PLS
; L162
LOAD      M14646	// R_3rd PP VC OFF PLS
OR        M14648	// R_3rd PP VC OFF
AND NOT   T1107	// R_3rd PP VC OFF TM
OUT       M14648	// R_3rd PP VC OFF
TON       T1107 D003030	// R_3rd PP VC OFF TM / T)PP VC OFF TM
// ========== 4th VACUUM ON/OFF ==========
; L165
LOAD      M14580	// R_P&P CYCLE RUN
AND       M14513	// R_P&P STEP#03
OR        M14842	// T)PP 4th VC ON
OR        M14650	// R_4th PP VC ON
AND NOT   M1451A	// R_P&P STEP#10
AND NOT   M14844	// T)PP 4th VC OFF
OUT       M14650	// R_4th PP VC ON
; L168
LOAD      M14650	// R_4th PP VC ON
OUT       P00166	// R_P&P 4th EJECT ON
; L169
LOAD      M14658	// R_4th PP VC OFF
OUT       P00167	// R_P&P 4th EJECT OFF
; L170
LOAD NOT  P00166	// R_P&P 4th EJECT ON
OUTP      M14656	// R_4th PP VC OFF PLS
; L171
LOAD      M14656	// R_4th PP VC OFF PLS
OR        M14658	// R_4th PP VC OFF
AND NOT   T1108	// R_4th PP VC OFF
OUT       M14658	// R_4th PP VC OFF
TON       T1108 D003030	// R_4th PP VC OFF / T)PP VC OFF TM

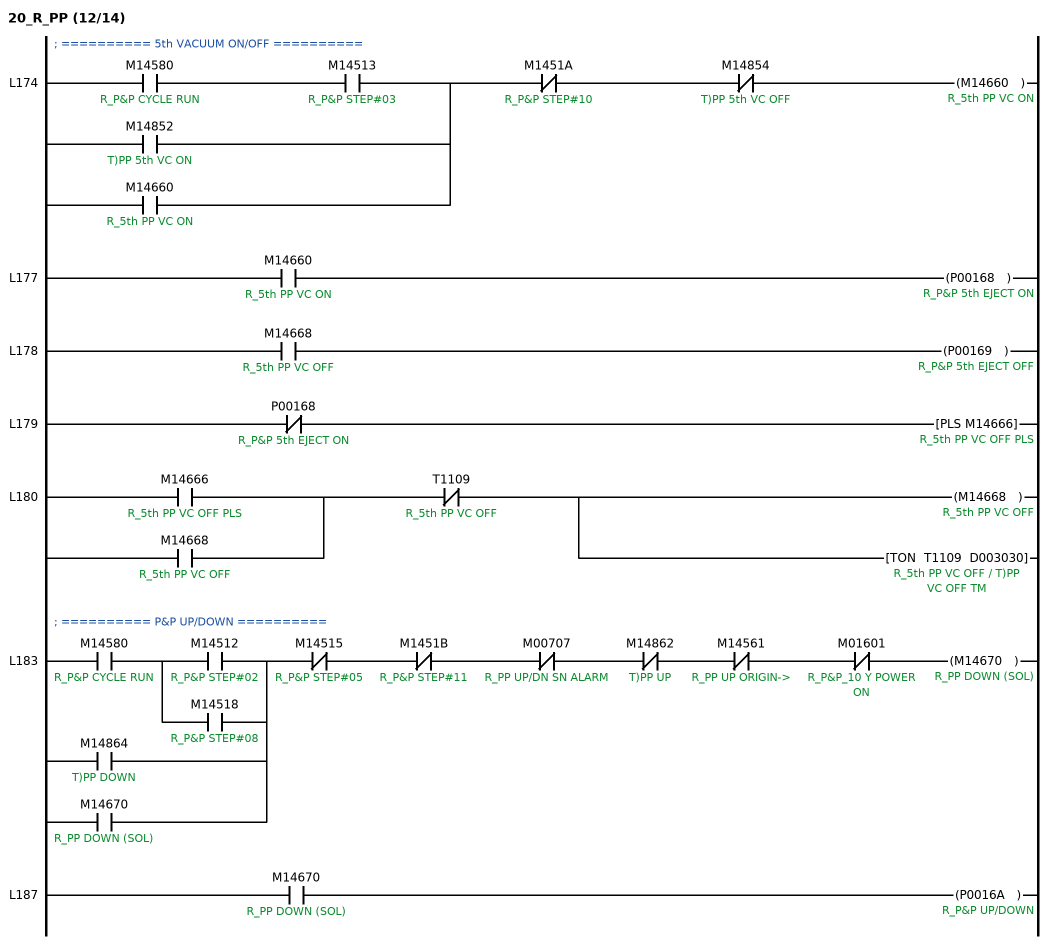
// ========== 5th VACUUM ON/OFF ==========
; L174
LOAD      M14580	// R_P&P CYCLE RUN
AND       M14513	// R_P&P STEP#03
OR        M14852	// T)PP 5th VC ON
OR        M14660	// R_5th PP VC ON
AND NOT   M1451A	// R_P&P STEP#10
AND NOT   M14854	// T)PP 5th VC OFF
OUT       M14660	// R_5th PP VC ON
; L177
LOAD      M14660	// R_5th PP VC ON
OUT       P00168	// R_P&P 5th EJECT ON
; L178
LOAD      M14668	// R_5th PP VC OFF
OUT       P00169	// R_P&P 5th EJECT OFF
; L179
LOAD NOT  P00168	// R_P&P 5th EJECT ON
OUTP      M14666	// R_5th PP VC OFF PLS
; L180
LOAD      M14666	// R_5th PP VC OFF PLS
OR        M14668	// R_5th PP VC OFF
AND NOT   T1109	// R_5th PP VC OFF
OUT       M14668	// R_5th PP VC OFF
TON       T1109 D003030	// R_5th PP VC OFF / T)PP VC OFF TM
// ========== P&P UP/DOWN ==========
; L183
LOAD      M14580	// R_P&P CYCLE RUN
LOAD      M14512	// R_P&P STEP#02
OR        M14518	// R_P&P STEP#08
AND LOAD
OR        M14864	// T)PP DOWN
OR        M14670	// R_PP DOWN (SOL)
AND NOT   M14515	// R_P&P STEP#05
AND NOT   M1451B	// R_P&P STEP#11
AND NOT   M00707	// R_PP UP/DN SN ALARM
AND NOT   M14862	// T)PP UP
AND NOT   M14561	// R_PP UP ORIGIN->
AND NOT   M01601	// R_P&P_10 Y POWER ON
OUT       M14670	// R_PP DOWN (SOL)
; L187
LOAD      M14670	// R_PP DOWN (SOL)
OUT       P0016A	// R_P&P UP/DOWN

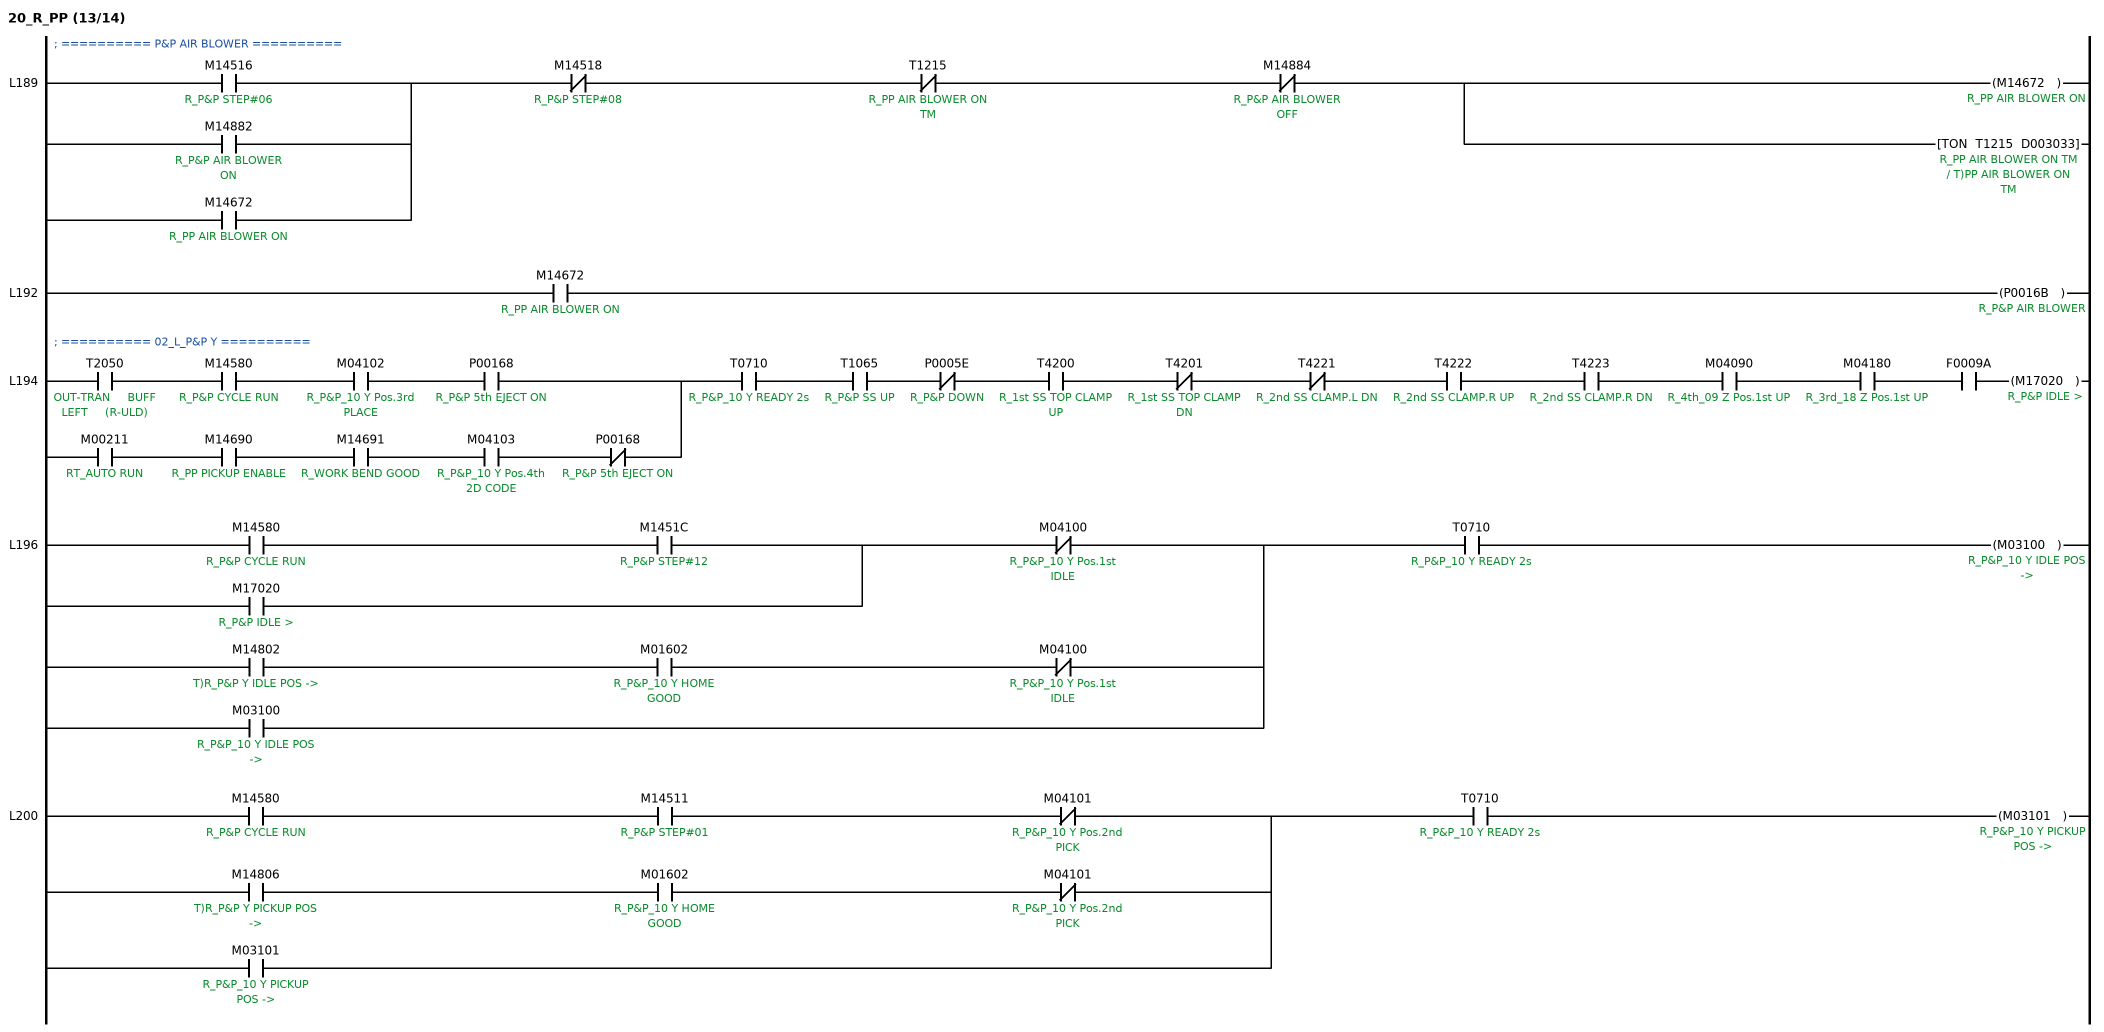
// ========== P&P AIR BLOWER ==========
; L189
LOAD      M14516	// R_P&P STEP#06
OR        M14882	// R_P&P AIR BLOWER ON
OR        M14672	// R_PP AIR BLOWER ON
AND NOT   M14518	// R_P&P STEP#08
AND NOT   T1215	// R_PP AIR BLOWER ON TM
AND NOT   M14884	// R_P&P AIR BLOWER OFF
OUT       M14672	// R_PP AIR BLOWER ON
TON       T1215 D003033	// R_PP AIR BLOWER ON TM / T)PP AIR BLOWER ON TM
; L192
LOAD      M14672	// R_PP AIR BLOWER ON
OUT       P0016B	// R_P&P AIR BLOWER
// ========== 02_L_P&P Y ==========
; L194
LOAD      T2050	// OUT-TRAN     BUFF     LEFT     (R-ULD)
AND       M14580	// R_P&P CYCLE RUN
AND       M04102	// R_P&P_10 Y Pos.3rd PLACE
AND       P00168	// R_P&P 5th EJECT ON
LOAD      M00211	// RT_AUTO RUN
AND       M14690	// R_PP PICKUP ENABLE
AND       M14691	// R_WORK BEND GOOD
AND       M04103	// R_P&P_10 Y Pos.4th 2D CODE
AND NOT   P00168	// R_P&P 5th EJECT ON
OR LOAD
AND       T0710	// R_P&P_10 Y READY 2s
AND       T1065	// R_P&P SS UP
AND NOT   P0005E	// R_P&P DOWN
AND       T4200	// R_1st SS TOP CLAMP UP
AND NOT   T4201	// R_1st SS TOP CLAMP DN
AND NOT   T4221	// R_2nd SS CLAMP.L DN
AND       T4222	// R_2nd SS CLAMP.R UP
AND       T4223	// R_2nd SS CLAMP.R DN
AND       M04090	// R_4th_09 Z Pos.1st UP
AND       M04180	// R_3rd_18 Z Pos.1st UP
AND       F0009A
OUT       M17020	// R_P&P IDLE >
; L196
LOAD      M14580	// R_P&P CYCLE RUN
AND       M1451C	// R_P&P STEP#12
OR        M17020	// R_P&P IDLE >
AND NOT   M04100	// R_P&P_10 Y Pos.1st IDLE
LOAD      M14802	// T)R_P&P Y IDLE POS ->
AND       M01602	// R_P&P_10 Y HOME GOOD
AND NOT   M04100	// R_P&P_10 Y Pos.1st IDLE
OR LOAD
OR        M03100	// R_P&P_10 Y IDLE POS ->
AND       T0710	// R_P&P_10 Y READY 2s
OUT       M03100	// R_P&P_10 Y IDLE POS ->
; L200
LOAD      M14580	// R_P&P CYCLE RUN
AND       M14511	// R_P&P STEP#01
AND NOT   M04101	// R_P&P_10 Y Pos.2nd PICK
LOAD      M14806	// T)R_P&P Y PICKUP POS ->
AND       M01602	// R_P&P_10 Y HOME GOOD
AND NOT   M04101	// R_P&P_10 Y Pos.2nd PICK
OR LOAD
OR        M03101	// R_P&P_10 Y PICKUP POS ->
AND       T0710	// R_P&P_10 Y READY 2s
OUT       M03101	// R_P&P_10 Y PICKUP POS ->

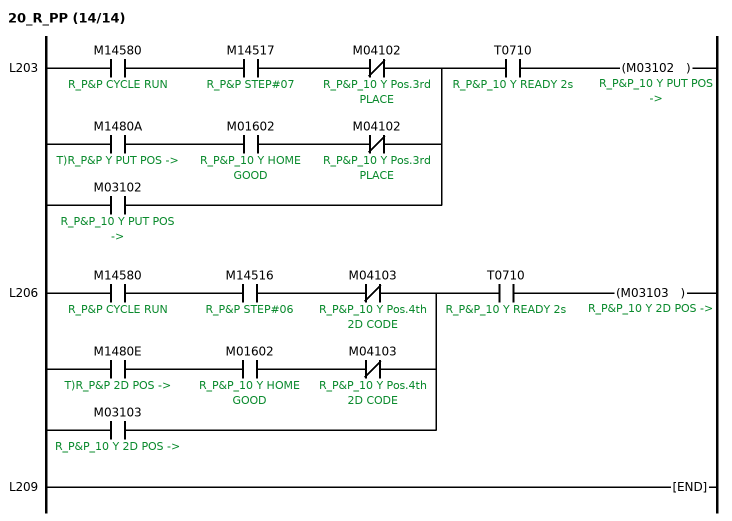
; L203
LOAD      M14580	// R_P&P CYCLE RUN
AND       M14517	// R_P&P STEP#07
AND NOT   M04102	// R_P&P_10 Y Pos.3rd PLACE
LOAD      M1480A	// T)R_P&P Y PUT POS ->
AND       M01602	// R_P&P_10 Y HOME GOOD
AND NOT   M04102	// R_P&P_10 Y Pos.3rd PLACE
OR LOAD
OR        M03102	// R_P&P_10 Y PUT POS ->
AND       T0710	// R_P&P_10 Y READY 2s
OUT       M03102	// R_P&P_10 Y PUT POS ->
; L206
LOAD      M14580	// R_P&P CYCLE RUN
AND       M14516	// R_P&P STEP#06
AND NOT   M04103	// R_P&P_10 Y Pos.4th 2D CODE
LOAD      M1480E	// T)R_P&P 2D POS ->
AND       M01602	// R_P&P_10 Y HOME GOOD
AND NOT   M04103	// R_P&P_10 Y Pos.4th 2D CODE
OR LOAD
OR        M03103	// R_P&P_10 Y 2D POS ->
AND       T0710	// R_P&P_10 Y READY 2s
OUT       M03103	// R_P&P_10 Y 2D POS ->
; L209
END

PROGRAM 30_IN_LR_BUFFER (task: ¨ö¨¬A¥ì CA¡¤I¡¾¡¿¡¤¡Í)

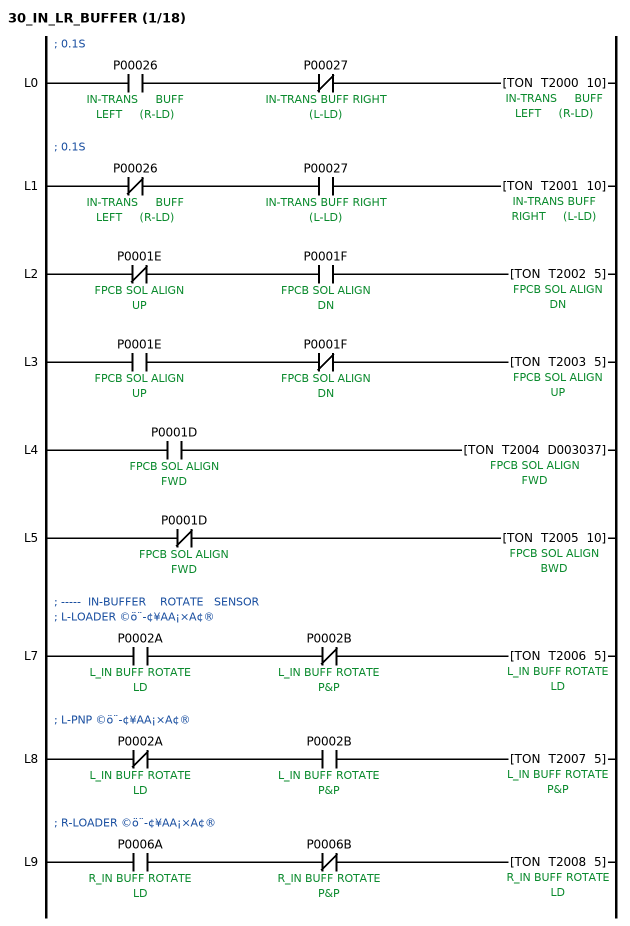
; L0
LOAD      P00026	// IN-TRANS     BUFF     LEFT     (R-LD)
AND NOT   P00027	// IN-TRANS BUFF RIGHT     (L-LD)
TON       T2000 10	// IN-TRANS     BUFF     LEFT     (R-LD)
// output comment: 0.1S
; L1
LOAD NOT  P00026	// IN-TRANS     BUFF     LEFT     (R-LD)
AND       P00027	// IN-TRANS BUFF RIGHT     (L-LD)
TON       T2001 10	// IN-TRANS BUFF RIGHT     (L-LD)
// output comment: 0.1S
; L2
LOAD NOT  P0001E	// FPCB SOL ALIGN         UP
AND       P0001F	// FPCB SOL ALIGN        DN
TON       T2002 5	// FPCB SOL ALIGN        DN
; L3
LOAD      P0001E	// FPCB SOL ALIGN         UP
AND NOT   P0001F	// FPCB SOL ALIGN        DN
TON       T2003 5	// FPCB SOL ALIGN         UP
; L4
LOAD      P0001D	// FPCB SOL ALIGN         FWD
TON       T2004 D003037	// FPCB SOL ALIGN         FWD
; L5
LOAD NOT  P0001D	// FPCB SOL ALIGN         FWD
TON       T2005 10	// FPCB SOL ALIGN         BWD
// -----  IN-BUFFER    ROTATE   SENSOR
; L7
LOAD      P0002A	// L_IN BUFF ROTATE     LD
AND NOT   P0002B	// L_IN BUFF ROTATE      P&P
TON       T2006 5	// L_IN BUFF ROTATE     LD
// output comment: L-LOADER ©ö¨­¢¥AA¡×A¢®
; L8
LOAD NOT  P0002A	// L_IN BUFF ROTATE     LD
AND       P0002B	// L_IN BUFF ROTATE      P&P
TON       T2007 5	// L_IN BUFF ROTATE      P&P
// output comment: L-PNP ©ö¨­¢¥AA¡×A¢®
; L9
LOAD      P0006A	// R_IN BUFF ROTATE      LD
AND NOT   P0006B	// R_IN BUFF ROTATE      P&P
TON       T2008 5	// R_IN BUFF ROTATE      LD
// output comment: R-LOADER ©ö¨­¢¥AA¡×A¢®

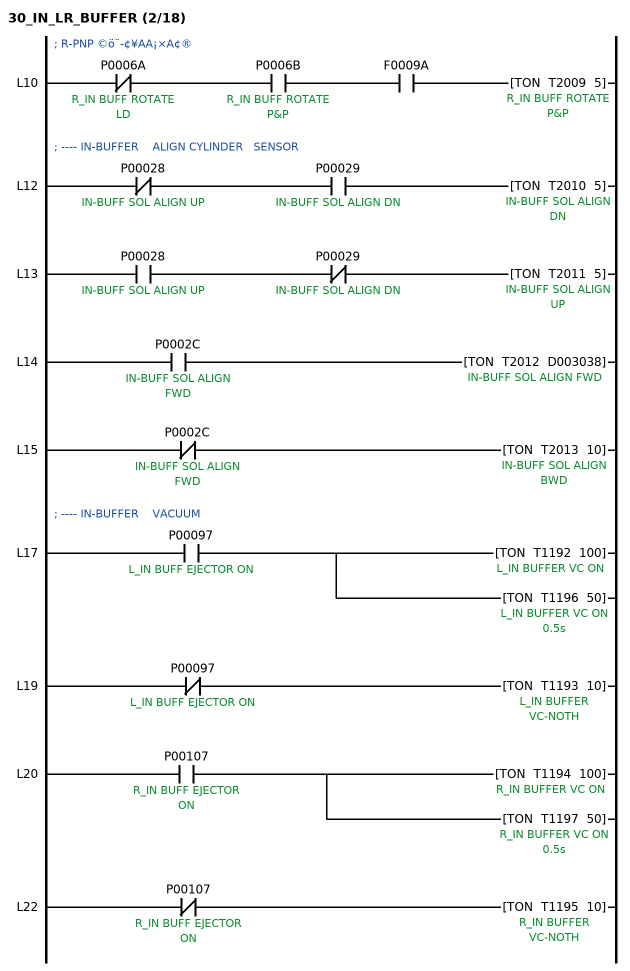
; L10
LOAD NOT  P0006A	// R_IN BUFF ROTATE      LD
AND       P0006B	// R_IN BUFF ROTATE      P&P
AND       F0009A
TON       T2009 5	// R_IN BUFF ROTATE      P&P
// output comment: R-PNP ©ö¨­¢¥AA¡×A¢®
// ---- IN-BUFFER    ALIGN CYLINDER   SENSOR
; L12
LOAD NOT  P00028	// IN-BUFF SOL ALIGN UP
AND       P00029	// IN-BUFF SOL ALIGN DN
TON       T2010 5	// IN-BUFF SOL ALIGN DN
; L13
LOAD      P00028	// IN-BUFF SOL ALIGN UP
AND NOT   P00029	// IN-BUFF SOL ALIGN DN
TON       T2011 5	// IN-BUFF SOL ALIGN UP
; L14
LOAD      P0002C	// IN-BUFF SOL ALIGN FWD
TON       T2012 D003038	// IN-BUFF SOL ALIGN FWD
; L15
LOAD NOT  P0002C	// IN-BUFF SOL ALIGN FWD
TON       T2013 10	// IN-BUFF SOL ALIGN BWD
// ---- IN-BUFFER    VACUUM
; L17
LOAD      P00097	// L_IN BUFF EJECTOR ON
TON       T1192 100	// L_IN BUFFER VC ON
TON       T1196 50	// L_IN BUFFER VC ON 0.5s
; L19
LOAD NOT  P00097	// L_IN BUFF EJECTOR ON
TON       T1193 10	// L_IN BUFFER VC-NOTH
; L20
LOAD      P00107	// R_IN BUFF EJECTOR ON
TON       T1194 100	// R_IN BUFFER VC ON
TON       T1197 50	// R_IN BUFFER VC ON 0.5s
; L22
LOAD NOT  P00107	// R_IN BUFF EJECTOR ON
TON       T1195 10	// R_IN BUFFER VC-NOTH

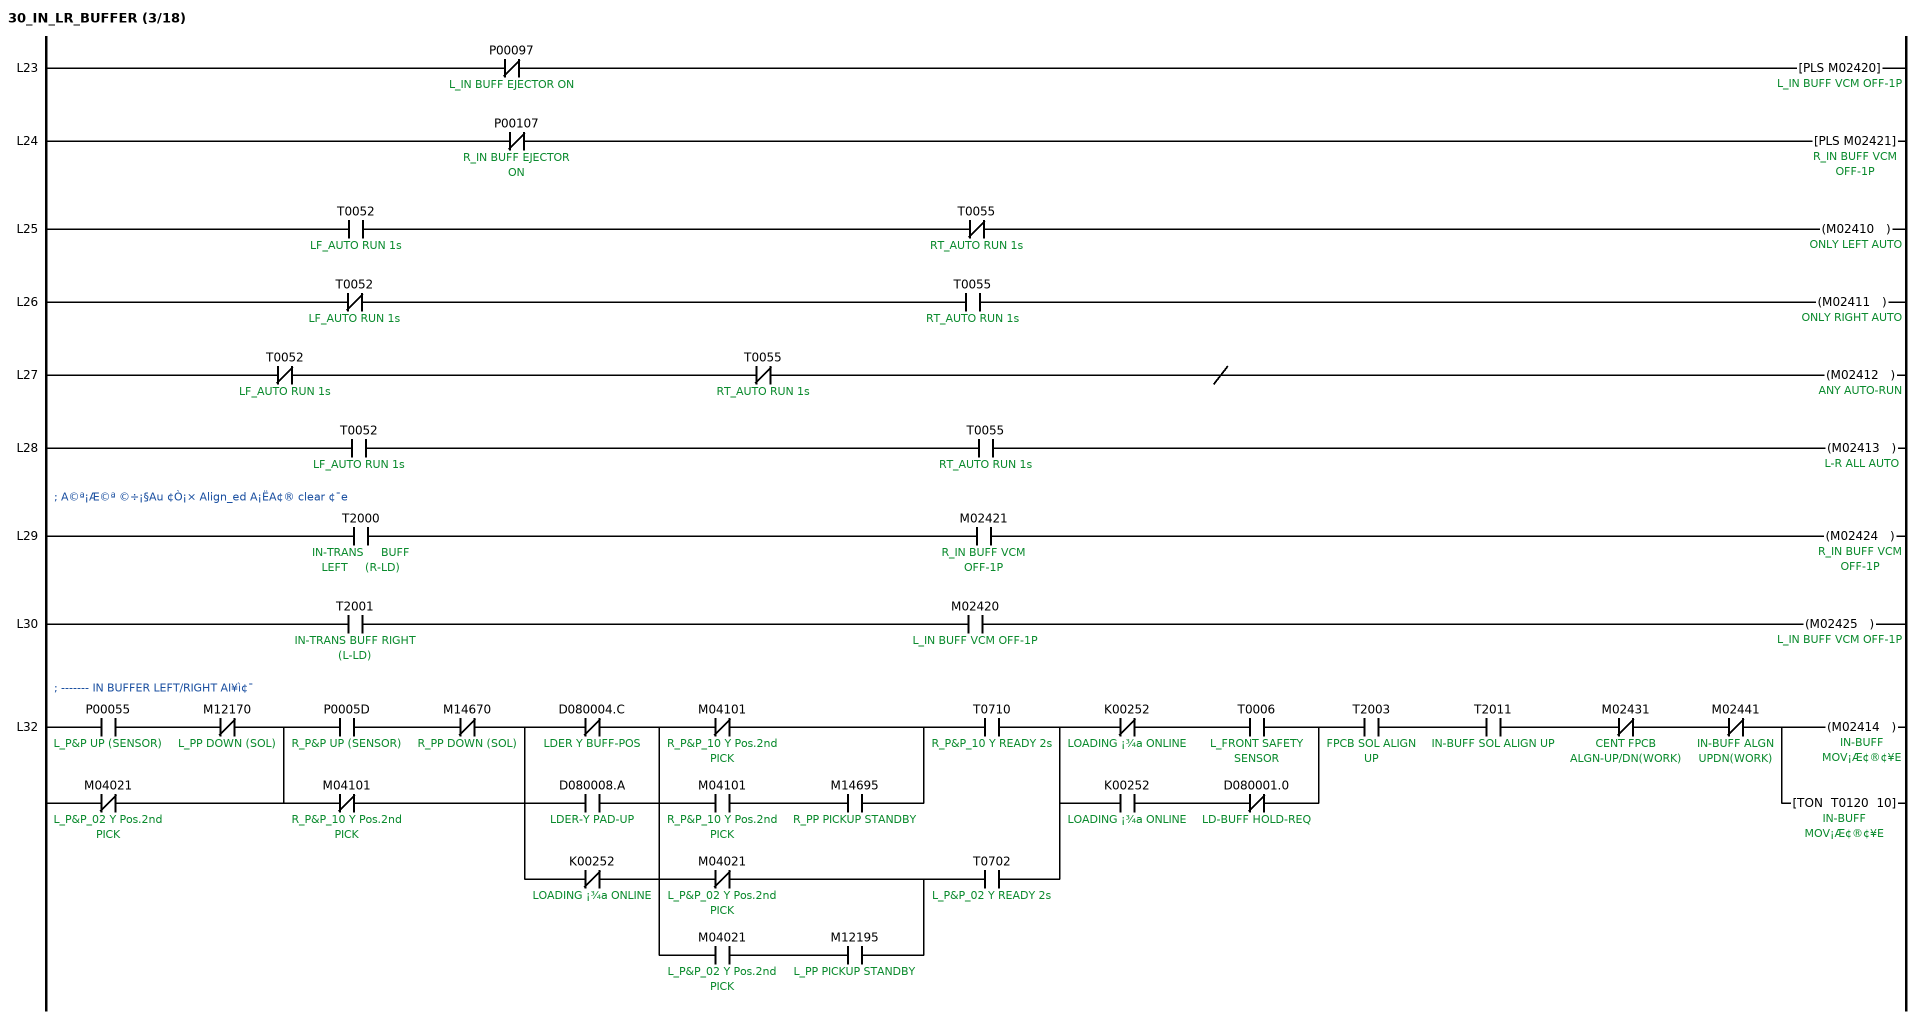
; L23
LOAD NOT  P00097	// L_IN BUFF EJECTOR ON
OUTP      M02420	// L_IN BUFF VCM OFF-1P
; L24
LOAD NOT  P00107	// R_IN BUFF EJECTOR ON
OUTP      M02421	// R_IN BUFF VCM OFF-1P
; L25
LOAD      T0052	// LF_AUTO RUN 1s
AND NOT   T0055	// RT_AUTO RUN 1s
OUT       M02410	// ONLY LEFT AUTO
; L26
LOAD NOT  T0052	// LF_AUTO RUN 1s
AND       T0055	// RT_AUTO RUN 1s
OUT       M02411	// ONLY RIGHT AUTO
; L27
LOAD NOT  T0052	// LF_AUTO RUN 1s
AND NOT   T0055	// RT_AUTO RUN 1s
NOT
OUT       M02412	// ANY AUTO-RUN
; L28
LOAD      T0052	// LF_AUTO RUN 1s
AND       T0055	// RT_AUTO RUN 1s
OUT       M02413	// L-R ALL AUTO
; L29
LOAD      T2000	// IN-TRANS     BUFF     LEFT     (R-LD)
AND       M02421	// R_IN BUFF VCM OFF-1P
OUT       M02424	// R_IN BUFF VCM OFF-1P
// output comment: A©ª¡Æ©ª ©÷¡§Au ¢Ò¡× Align_ed A¡ËA¢® clear ¢¯e
; L30
LOAD      T2001	// IN-TRANS BUFF RIGHT     (L-LD)
AND       M02420	// L_IN BUFF VCM OFF-1P
OUT       M02425	// L_IN BUFF VCM OFF-1P
// ------- IN BUFFER LEFT/RIGHT AI¥ì¢¯
; L32
LOAD      P00055	// L_P&P UP (SENSOR)
AND NOT   M12170	// L_PP DOWN (SOL)
OR NOT    M04021	// L_P&P_02 Y Pos.2nd PICK
LOAD      P0005D	// R_P&P UP (SENSOR)
AND NOT   M14670	// R_PP DOWN (SOL)
OR NOT    M04101	// R_P&P_10 Y Pos.2nd PICK
AND LOAD
LOAD NOT  D080004.C	// LDER Y BUFF-POS
OR        D080008.A	// LDER-Y PAD-UP
OR NOT    K00252	// LOADING ¡¾a ONLINE
AND LOAD
LOAD NOT  M04101	// R_P&P_10 Y Pos.2nd PICK
LOAD      M04101	// R_P&P_10 Y Pos.2nd PICK
AND       M14695	// R_PP PICKUP STANDBY
OR LOAD
AND       T0710	// R_P&P_10 Y READY 2s
LOAD NOT  M04021	// L_P&P_02 Y Pos.2nd PICK
LOAD      M04021	// L_P&P_02 Y Pos.2nd PICK
AND       M12195	// L_PP PICKUP STANDBY
OR LOAD
AND       T0702	// L_P&P_02 Y READY 2s
OR LOAD
AND LOAD
LOAD NOT  K00252	// LOADING ¡¾a ONLINE
AND       T0006	// L_FRONT SAFETY SENSOR
LOAD      K00252	// LOADING ¡¾a ONLINE
AND NOT   D080001.0	// LD-BUFF HOLD-REQ
OR LOAD
AND LOAD
AND       T2003	// FPCB SOL ALIGN         UP
AND       T2011	// IN-BUFF SOL ALIGN UP
AND NOT   M02431	// CENT FPCB ALGN-UP/DN(WORK)
AND NOT   M02441	// IN-BUFF ALGN UPDN(WORK)
OUT       M02414	// IN-BUFF MOV¡Æ¢®¢¥E
TON       T0120 10	// IN-BUFF MOV¡Æ¢®¢¥E

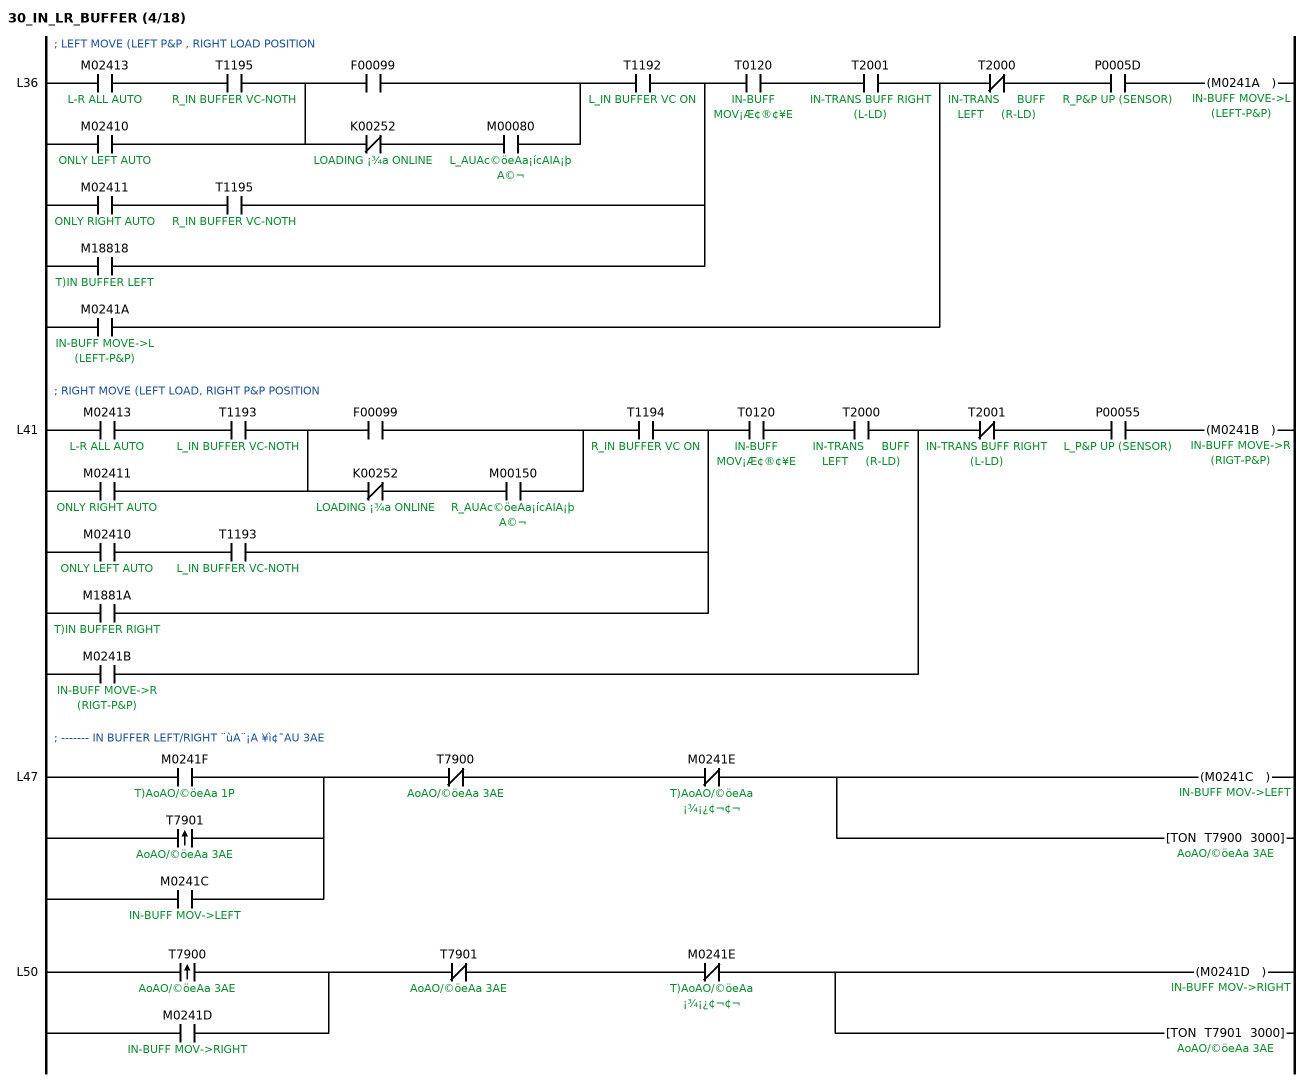
; L36
LOAD      M02413	// L-R ALL AUTO
AND       T1195	// R_IN BUFFER VC-NOTH
OR        M02410	// ONLY LEFT AUTO
LOAD      F00099
LOAD NOT  K00252	// LOADING ¡¾a ONLINE
AND       M00080	// L_AUAc©öeAa¡ícAIA¡þA©¬
OR LOAD
AND LOAD
AND       T1192	// L_IN BUFFER VC ON
LOAD      M02411	// ONLY RIGHT AUTO
AND       T1195	// R_IN BUFFER VC-NOTH
OR LOAD
OR        M18818	// T)IN BUFFER LEFT
AND       T0120	// IN-BUFF MOV¡Æ¢®¢¥E
AND       T2001	// IN-TRANS BUFF RIGHT     (L-LD)
OR        M0241A	// IN-BUFF MOVE->L (LEFT-P&P)
AND NOT   T2000	// IN-TRANS     BUFF     LEFT     (R-LD)
AND       P0005D	// R_P&P UP (SENSOR)
OUT       M0241A	// IN-BUFF MOVE->L (LEFT-P&P)
// output comment: LEFT MOVE (LEFT P&P , RIGHT LOAD POSITION
; L41
LOAD      M02413	// L-R ALL AUTO
AND       T1193	// L_IN BUFFER VC-NOTH
OR        M02411	// ONLY RIGHT AUTO
LOAD      F00099
LOAD NOT  K00252	// LOADING ¡¾a ONLINE
AND       M00150	// R_AUAc©öeAa¡ícAIA¡þA©¬
OR LOAD
AND LOAD
AND       T1194	// R_IN BUFFER VC ON
LOAD      M02410	// ONLY LEFT AUTO
AND       T1193	// L_IN BUFFER VC-NOTH
OR LOAD
OR        M1881A	// T)IN BUFFER RIGHT
AND       T0120	// IN-BUFF MOV¡Æ¢®¢¥E
AND       T2000	// IN-TRANS     BUFF     LEFT     (R-LD)
OR        M0241B	// IN-BUFF MOVE->R (RIGT-P&P)
AND NOT   T2001	// IN-TRANS BUFF RIGHT     (L-LD)
AND       P00055	// L_P&P UP (SENSOR)
OUT       M0241B	// IN-BUFF MOVE->R (RIGT-P&P)
// output comment: RIGHT MOVE (LEFT LOAD, RIGHT P&P POSITION
// ------- IN BUFFER LEFT/RIGHT ¨ùA¨¡A ¥ì¢¯AU 3AE
; L47
LOAD      M0241F	// T)AoAO/©öeAa 1P
ORP       T7901	// AoAO/©öeAa 3AE
OR        M0241C	// IN-BUFF MOV->LEFT
AND NOT   T7900	// AoAO/©öeAa 3AE
AND NOT   M0241E	// T)AoAO/©öeAa ¡¾¡¿¢¬¢¬
OUT       M0241C	// IN-BUFF MOV->LEFT
TON       T7900 3000	// AoAO/©öeAa 3AE
; L50
LOADP     T7900	// AoAO/©öeAa 3AE
OR        M0241D	// IN-BUFF MOV->RIGHT
AND NOT   T7901	// AoAO/©öeAa 3AE
AND NOT   M0241E	// T)AoAO/©öeAa ¡¾¡¿¢¬¢¬
OUT       M0241D	// IN-BUFF MOV->RIGHT
TON       T7901 3000	// AoAO/©öeAa 3AE

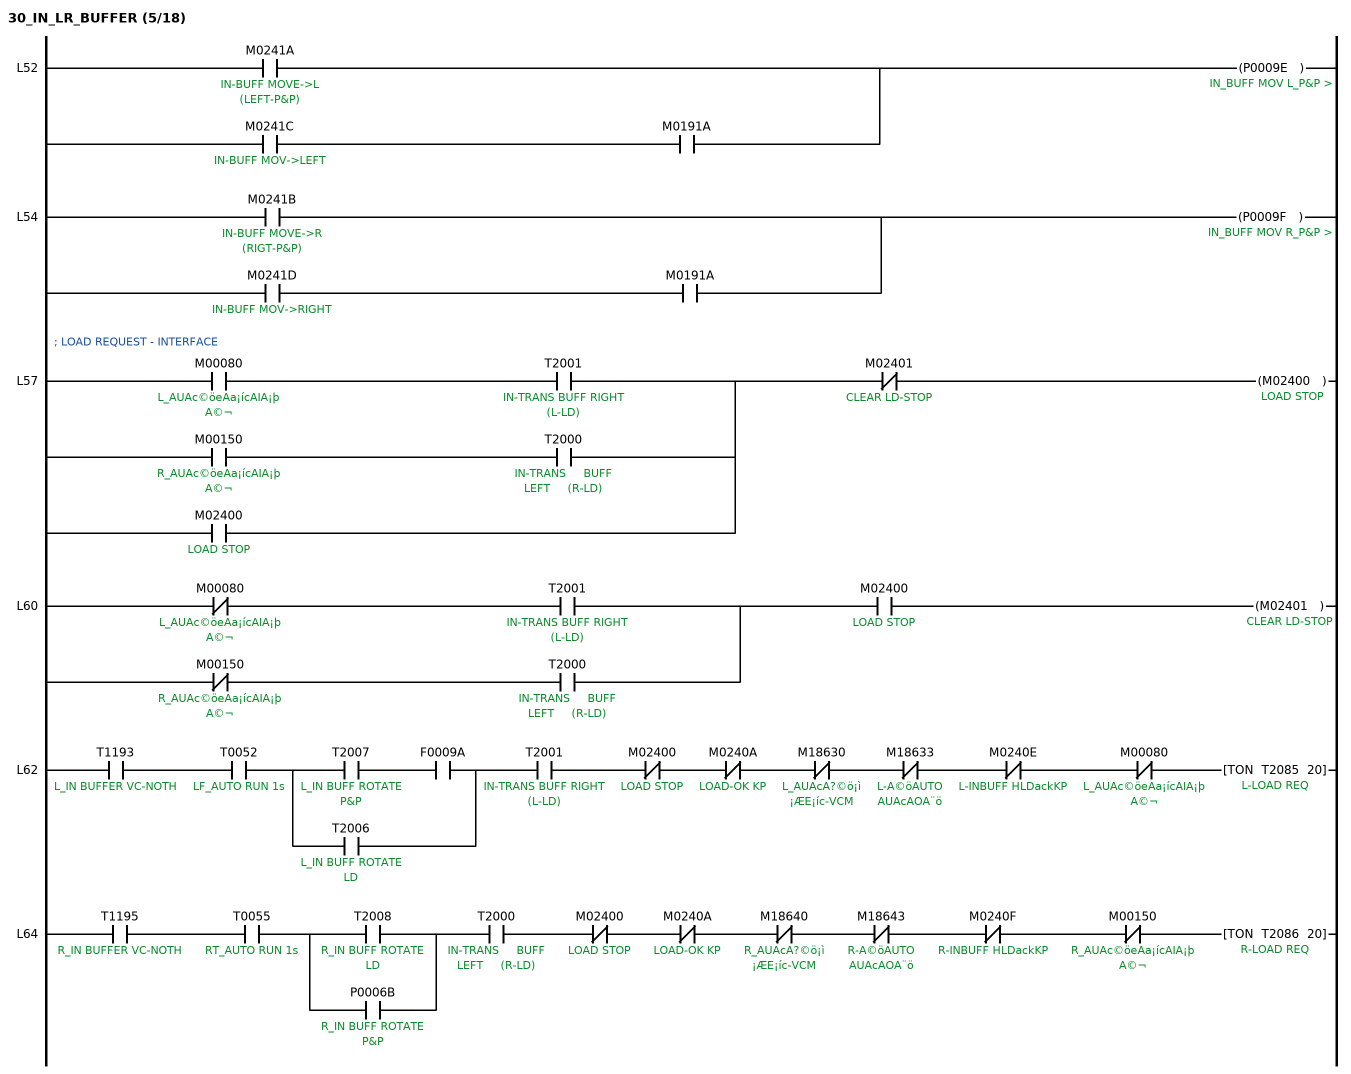
; L52
LOAD      M0241A	// IN-BUFF MOVE->L (LEFT-P&P)
LOAD      M0241C	// IN-BUFF MOV->LEFT
AND       M0191A
OR LOAD
OUT       P0009E	// IN_BUFF MOV L_P&P >
; L54
LOAD      M0241B	// IN-BUFF MOVE->R (RIGT-P&P)
LOAD      M0241D	// IN-BUFF MOV->RIGHT
AND       M0191A
OR LOAD
OUT       P0009F	// IN_BUFF MOV R_P&P >
// LOAD REQUEST - INTERFACE
; L57
LOAD      M00080	// L_AUAc©öeAa¡ícAIA¡þA©¬
AND       T2001	// IN-TRANS BUFF RIGHT     (L-LD)
LOAD      M00150	// R_AUAc©öeAa¡ícAIA¡þA©¬
AND       T2000	// IN-TRANS     BUFF     LEFT     (R-LD)
OR LOAD
OR        M02400	// LOAD STOP
AND NOT   M02401	// CLEAR LD-STOP
OUT       M02400	// LOAD STOP
; L60
LOAD NOT  M00080	// L_AUAc©öeAa¡ícAIA¡þA©¬
AND       T2001	// IN-TRANS BUFF RIGHT     (L-LD)
LOAD NOT  M00150	// R_AUAc©öeAa¡ícAIA¡þA©¬
AND       T2000	// IN-TRANS     BUFF     LEFT     (R-LD)
OR LOAD
AND       M02400	// LOAD STOP
OUT       M02401	// CLEAR LD-STOP
; L62
LOAD      T1193	// L_IN BUFFER VC-NOTH
AND       T0052	// LF_AUTO RUN 1s
LOAD      T2007	// L_IN BUFF ROTATE      P&P
AND       F0009A
OR        T2006	// L_IN BUFF ROTATE     LD
AND LOAD
AND       T2001	// IN-TRANS BUFF RIGHT     (L-LD)
AND NOT   M02400	// LOAD STOP
AND NOT   M0240A	// LOAD-OK KP
AND NOT   M18630	// L_AUAcA?©ö¡ì ¡ÆE¡íc-VCM
AND NOT   M18633	// L-A©öAUTO AUAcAOA¨ö
AND NOT   M0240E	// L-INBUFF HLDackKP
AND NOT   M00080	// L_AUAc©öeAa¡ícAIA¡þA©¬
TON       T2085 20	// L-LOAD REQ
; L64
LOAD      T1195	// R_IN BUFFER VC-NOTH
AND       T0055	// RT_AUTO RUN 1s
LOAD      T2008	// R_IN BUFF ROTATE      LD
OR        P0006B	// R_IN BUFF ROTATE      P&P
AND LOAD
AND       T2000	// IN-TRANS     BUFF     LEFT     (R-LD)
AND NOT   M02400	// LOAD STOP
AND NOT   M0240A	// LOAD-OK KP
AND NOT   M18640	// R_AUAcA?©ö¡ì ¡ÆE¡íc-VCM
AND NOT   M18643	// R-A©öAUTO AUAcAOA¨ö
AND NOT   M0240F	// R-INBUFF HLDackKP
AND NOT   M00150	// R_AUAc©öeAa¡ícAIA¡þA©¬
TON       T2086 20	// R-LOAD REQ

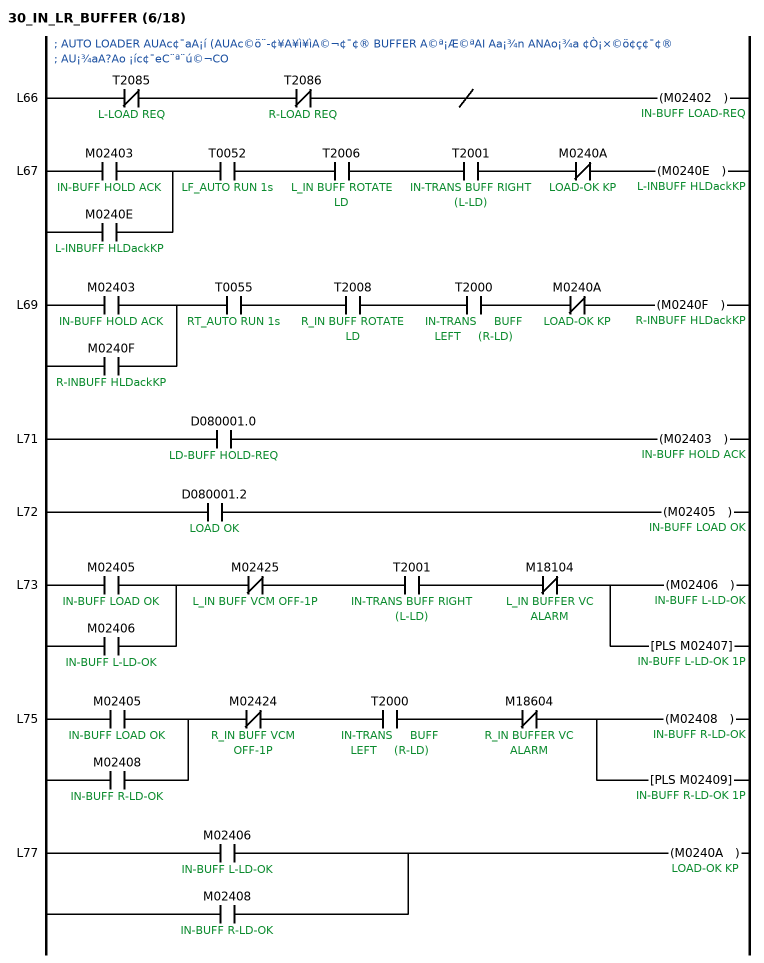
; L66
LOAD NOT  T2085	// L-LOAD REQ
AND NOT   T2086	// R-LOAD REQ
NOT
OUT       M02402	// IN-BUFF LOAD-REQ
// output comment: AUTO LOADER AUAc¢¯aA¡í (AUAc©ö¨­¢¥A¥ì¥ìA©¬¢¯¢® BUFFER A©ª¡Æ©ªAI Aa¡¾n ANAo¡¾a ¢Ò¡×©ö¢ç¢¯¢® AU¡¾aA?Ao ¡íc¢¯eC¨ª¨ú©¬CO
; L67
LOAD      M02403	// IN-BUFF HOLD ACK
OR        M0240E	// L-INBUFF HLDackKP
AND       T0052	// LF_AUTO RUN 1s
AND       T2006	// L_IN BUFF ROTATE     LD
AND       T2001	// IN-TRANS BUFF RIGHT     (L-LD)
AND NOT   M0240A	// LOAD-OK KP
OUT       M0240E	// L-INBUFF HLDackKP
; L69
LOAD      M02403	// IN-BUFF HOLD ACK
OR        M0240F	// R-INBUFF HLDackKP
AND       T0055	// RT_AUTO RUN 1s
AND       T2008	// R_IN BUFF ROTATE      LD
AND       T2000	// IN-TRANS     BUFF     LEFT     (R-LD)
AND NOT   M0240A	// LOAD-OK KP
OUT       M0240F	// R-INBUFF HLDackKP
; L71
LOAD      D080001.0	// LD-BUFF HOLD-REQ
OUT       M02403	// IN-BUFF HOLD ACK
; L72
LOAD      D080001.2	// LOAD OK
OUT       M02405	// IN-BUFF LOAD OK
; L73
LOAD      M02405	// IN-BUFF LOAD OK
OR        M02406	// IN-BUFF L-LD-OK
AND NOT   M02425	// L_IN BUFF VCM OFF-1P
AND       T2001	// IN-TRANS BUFF RIGHT     (L-LD)
AND NOT   M18104	// L_IN BUFFER VC ALARM
OUT       M02406	// IN-BUFF L-LD-OK
OUTP      M02407	// IN-BUFF L-LD-OK 1P
; L75
LOAD      M02405	// IN-BUFF LOAD OK
OR        M02408	// IN-BUFF R-LD-OK
AND NOT   M02424	// R_IN BUFF VCM OFF-1P
AND       T2000	// IN-TRANS     BUFF     LEFT     (R-LD)
AND NOT   M18604	// R_IN BUFFER VC ALARM
OUT       M02408	// IN-BUFF R-LD-OK
OUTP      M02409	// IN-BUFF R-LD-OK 1P
; L77
LOAD      M02406	// IN-BUFF L-LD-OK
OR        M02408	// IN-BUFF R-LD-OK
OUT       M0240A	// LOAD-OK KP

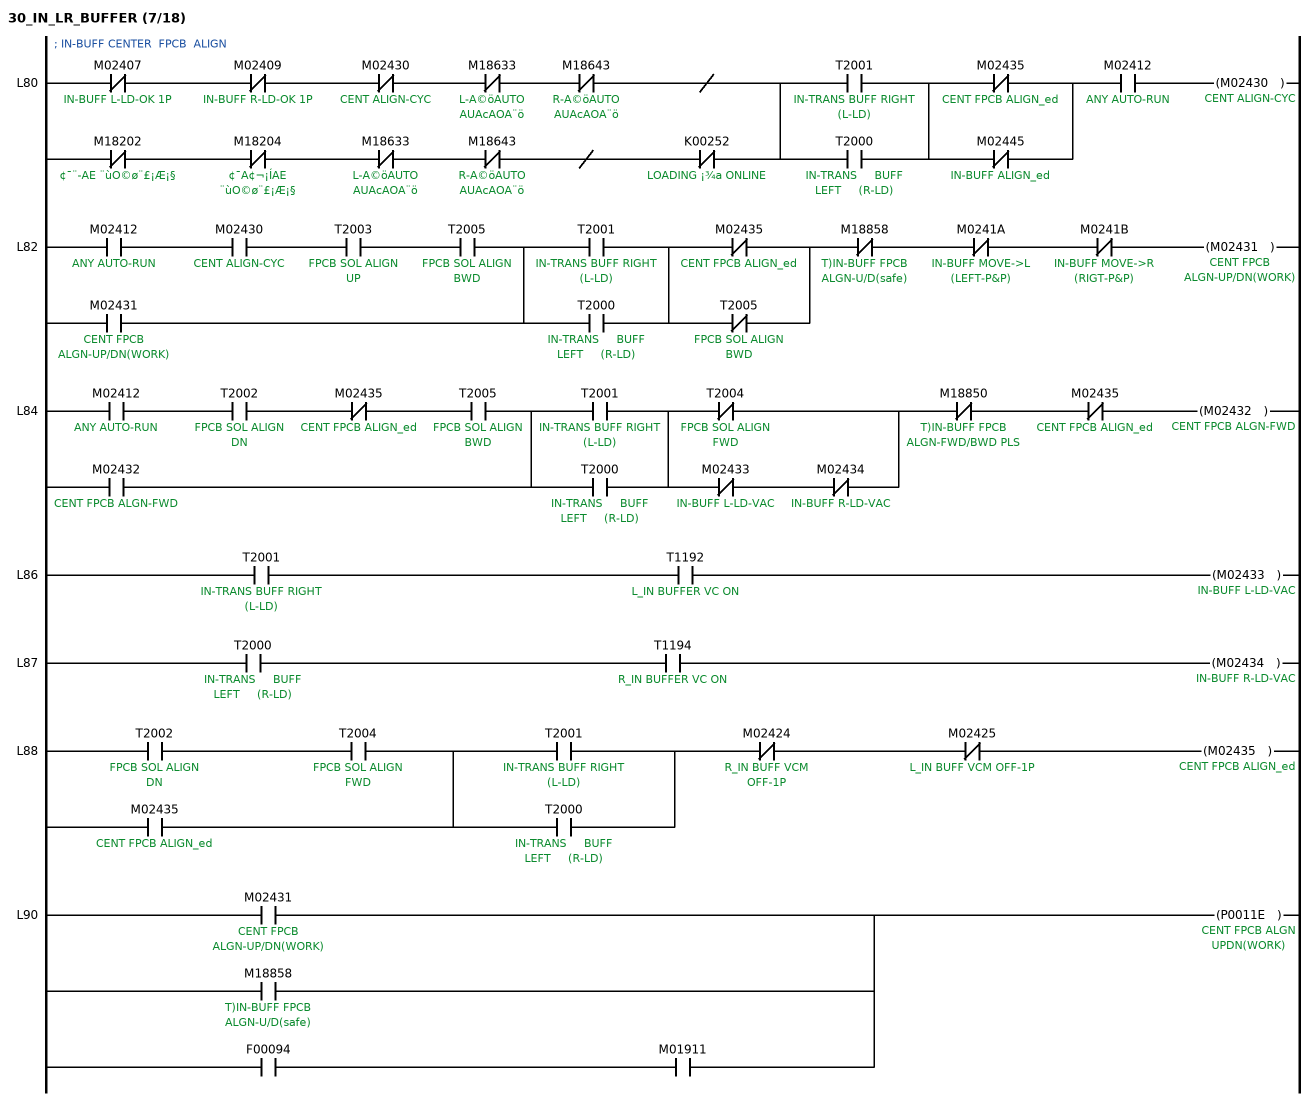
// IN-BUFF CENTER  FPCB  ALIGN
; L80
LOAD NOT  M02407	// IN-BUFF L-LD-OK 1P
AND NOT   M02409	// IN-BUFF R-LD-OK 1P
AND NOT   M02430	// CENT ALIGN-CYC
AND NOT   M18633	// L-A©öAUTO AUAcAOA¨ö
AND NOT   M18643	// R-A©öAUTO AUAcAOA¨ö
NOT
LOAD NOT  M18202	// ¢¯¨­AE ¨ùO©ø¨£¡Æ¡§
AND NOT   M18204	// ¢¯A¢¬¡ÍAE ¨ùO©ø¨£¡Æ¡§
AND NOT   M18633	// L-A©öAUTO AUAcAOA¨ö
AND NOT   M18643	// R-A©öAUTO AUAcAOA¨ö
NOT
AND NOT   K00252	// LOADING ¡¾a ONLINE
OR LOAD
LOAD      T2001	// IN-TRANS BUFF RIGHT     (L-LD)
OR        T2000	// IN-TRANS     BUFF     LEFT     (R-LD)
AND LOAD
LOAD NOT  M02435	// CENT FPCB ALIGN_ed
OR NOT    M02445	// IN-BUFF ALIGN_ed
AND LOAD
AND       M02412	// ANY AUTO-RUN
OUT       M02430	// CENT ALIGN-CYC
; L82
LOAD      M02412	// ANY AUTO-RUN
AND       M02430	// CENT ALIGN-CYC
AND       T2003	// FPCB SOL ALIGN         UP
AND       T2005	// FPCB SOL ALIGN         BWD
OR        M02431	// CENT FPCB ALGN-UP/DN(WORK)
LOAD      T2001	// IN-TRANS BUFF RIGHT     (L-LD)
OR        T2000	// IN-TRANS     BUFF     LEFT     (R-LD)
AND LOAD
LOAD NOT  M02435	// CENT FPCB ALIGN_ed
OR NOT    T2005	// FPCB SOL ALIGN         BWD
AND LOAD
AND NOT   M18858	// T)IN-BUFF FPCB ALGN-U/D(safe)
AND NOT   M0241A	// IN-BUFF MOVE->L (LEFT-P&P)
AND NOT   M0241B	// IN-BUFF MOVE->R (RIGT-P&P)
OUT       M02431	// CENT FPCB ALGN-UP/DN(WORK)
; L84
LOAD      M02412	// ANY AUTO-RUN
AND       T2002	// FPCB SOL ALIGN        DN
AND NOT   M02435	// CENT FPCB ALIGN_ed
AND       T2005	// FPCB SOL ALIGN         BWD
OR        M02432	// CENT FPCB ALGN-FWD
LOAD      T2001	// IN-TRANS BUFF RIGHT     (L-LD)
OR        T2000	// IN-TRANS     BUFF     LEFT     (R-LD)
AND LOAD
LOAD NOT  T2004	// FPCB SOL ALIGN         FWD
LOAD NOT  M02433	// IN-BUFF L-LD-VAC
AND NOT   M02434	// IN-BUFF R-LD-VAC
OR LOAD
AND LOAD
AND NOT   M18850	// T)IN-BUFF FPCB ALGN-FWD/BWD PLS
AND NOT   M02435	// CENT FPCB ALIGN_ed
OUT       M02432	// CENT FPCB ALGN-FWD
; L86
LOAD      T2001	// IN-TRANS BUFF RIGHT     (L-LD)
AND       T1192	// L_IN BUFFER VC ON
OUT       M02433	// IN-BUFF L-LD-VAC
; L87
LOAD      T2000	// IN-TRANS     BUFF     LEFT     (R-LD)
AND       T1194	// R_IN BUFFER VC ON
OUT       M02434	// IN-BUFF R-LD-VAC
; L88
LOAD      T2002	// FPCB SOL ALIGN        DN
AND       T2004	// FPCB SOL ALIGN         FWD
OR        M02435	// CENT FPCB ALIGN_ed
LOAD      T2001	// IN-TRANS BUFF RIGHT     (L-LD)
OR        T2000	// IN-TRANS     BUFF     LEFT     (R-LD)
AND LOAD
AND NOT   M02424	// R_IN BUFF VCM OFF-1P
AND NOT   M02425	// L_IN BUFF VCM OFF-1P
OUT       M02435	// CENT FPCB ALIGN_ed
; L90
LOAD      M02431	// CENT FPCB ALGN-UP/DN(WORK)
OR        M18858	// T)IN-BUFF FPCB ALGN-U/D(safe)
LOAD      F00094
AND       M01911
OR LOAD
OUT       P0011E	// CENT FPCB ALGN UPDN(WORK)

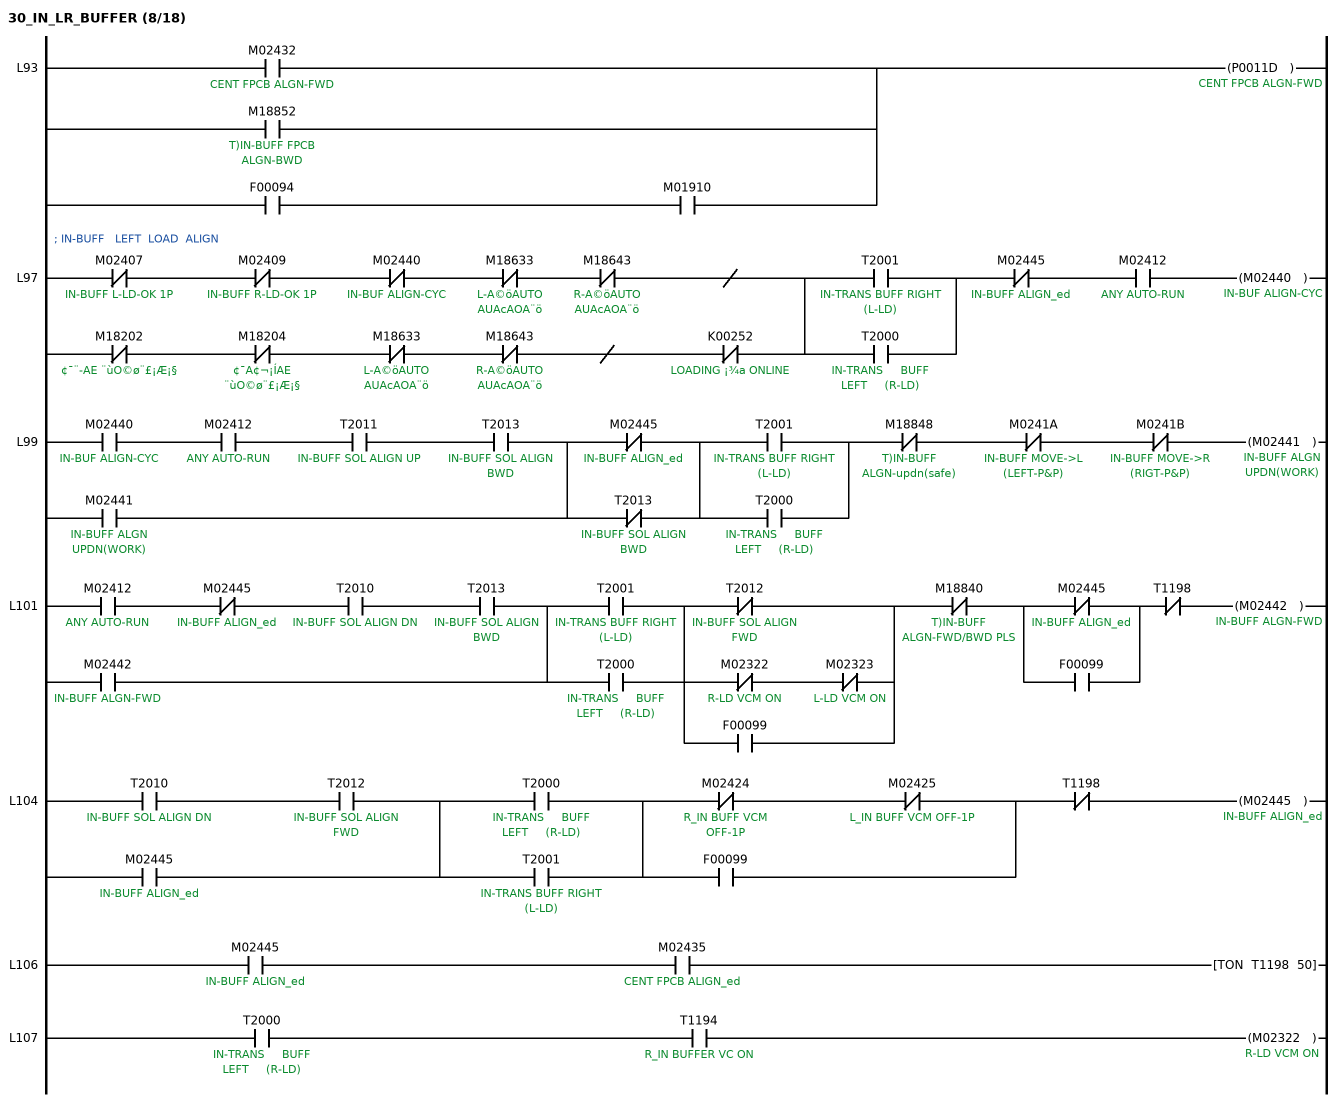
; L93
LOAD      M02432	// CENT FPCB ALGN-FWD
OR        M18852	// T)IN-BUFF FPCB ALGN-BWD
LOAD      F00094
AND       M01910
OR LOAD
OUT       P0011D	// CENT FPCB ALGN-FWD
// IN-BUFF   LEFT  LOAD  ALIGN
; L97
LOAD NOT  M02407	// IN-BUFF L-LD-OK 1P
AND NOT   M02409	// IN-BUFF R-LD-OK 1P
AND NOT   M02440	// IN-BUF ALIGN-CYC
AND NOT   M18633	// L-A©öAUTO AUAcAOA¨ö
AND NOT   M18643	// R-A©öAUTO AUAcAOA¨ö
NOT
LOAD NOT  M18202	// ¢¯¨­AE ¨ùO©ø¨£¡Æ¡§
AND NOT   M18204	// ¢¯A¢¬¡ÍAE ¨ùO©ø¨£¡Æ¡§
AND NOT   M18633	// L-A©öAUTO AUAcAOA¨ö
AND NOT   M18643	// R-A©öAUTO AUAcAOA¨ö
NOT
AND NOT   K00252	// LOADING ¡¾a ONLINE
OR LOAD
LOAD      T2001	// IN-TRANS BUFF RIGHT     (L-LD)
OR        T2000	// IN-TRANS     BUFF     LEFT     (R-LD)
AND LOAD
AND NOT   M02445	// IN-BUFF ALIGN_ed
AND       M02412	// ANY AUTO-RUN
OUT       M02440	// IN-BUF ALIGN-CYC
; L99
LOAD      M02440	// IN-BUF ALIGN-CYC
AND       M02412	// ANY AUTO-RUN
AND       T2011	// IN-BUFF SOL ALIGN UP
AND       T2013	// IN-BUFF SOL ALIGN BWD
OR        M02441	// IN-BUFF ALGN UPDN(WORK)
LOAD NOT  M02445	// IN-BUFF ALIGN_ed
OR NOT    T2013	// IN-BUFF SOL ALIGN BWD
AND LOAD
LOAD      T2001	// IN-TRANS BUFF RIGHT     (L-LD)
OR        T2000	// IN-TRANS     BUFF     LEFT     (R-LD)
AND LOAD
AND NOT   M18848	// T)IN-BUFF ALGN-updn(safe)
AND NOT   M0241A	// IN-BUFF MOVE->L (LEFT-P&P)
AND NOT   M0241B	// IN-BUFF MOVE->R (RIGT-P&P)
OUT       M02441	// IN-BUFF ALGN UPDN(WORK)
; L101
LOAD      M02412	// ANY AUTO-RUN
AND NOT   M02445	// IN-BUFF ALIGN_ed
AND       T2010	// IN-BUFF SOL ALIGN DN
AND       T2013	// IN-BUFF SOL ALIGN BWD
OR        M02442	// IN-BUFF ALGN-FWD
LOAD      T2001	// IN-TRANS BUFF RIGHT     (L-LD)
OR        T2000	// IN-TRANS     BUFF     LEFT     (R-LD)
AND LOAD
LOAD NOT  T2012	// IN-BUFF SOL ALIGN FWD
LOAD NOT  M02322	// R-LD VCM ON
AND NOT   M02323	// L-LD VCM ON
OR LOAD
OR        F00099
AND LOAD
AND NOT   M18840	// T)IN-BUFF ALGN-FWD/BWD PLS
LOAD NOT  M02445	// IN-BUFF ALIGN_ed
OR        F00099
AND LOAD
AND NOT   T1198
OUT       M02442	// IN-BUFF ALGN-FWD
; L104
LOAD      T2010	// IN-BUFF SOL ALIGN DN
AND       T2012	// IN-BUFF SOL ALIGN FWD
OR        M02445	// IN-BUFF ALIGN_ed
LOAD      T2000	// IN-TRANS     BUFF     LEFT     (R-LD)
OR        T2001	// IN-TRANS BUFF RIGHT     (L-LD)
AND LOAD
LOAD NOT  M02424	// R_IN BUFF VCM OFF-1P
AND NOT   M02425	// L_IN BUFF VCM OFF-1P
OR        F00099
AND LOAD
AND NOT   T1198
OUT       M02445	// IN-BUFF ALIGN_ed
; L106
LOAD      M02445	// IN-BUFF ALIGN_ed
AND       M02435	// CENT FPCB ALIGN_ed
TON       T1198 50
; L107
LOAD      T2000	// IN-TRANS     BUFF     LEFT     (R-LD)
AND       T1194	// R_IN BUFFER VC ON
OUT       M02322	// R-LD VCM ON

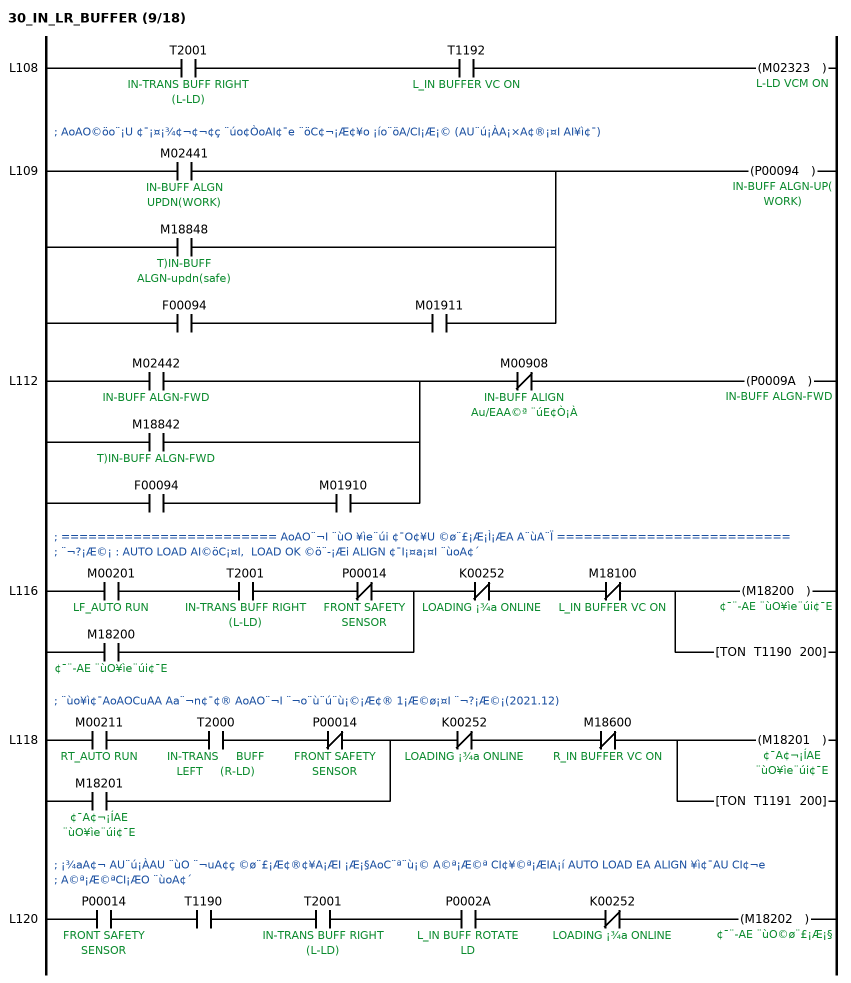
; L108
LOAD      T2001	// IN-TRANS BUFF RIGHT     (L-LD)
AND       T1192	// L_IN BUFFER VC ON
OUT       M02323	// L-LD VCM ON
; L109
LOAD      M02441	// IN-BUFF ALGN UPDN(WORK)
OR        M18848	// T)IN-BUFF ALGN-updn(safe)
LOAD      F00094
AND       M01911
OR LOAD
OUT       P00094	// IN-BUFF ALGN-UP(WORK)
// output comment: AoAO©öo¨¡U ¢¯¡¤¡¾¢¬¢¬¢ç ¨úo¢ÒoAI¢¯e ¨öC¢¬¡Æ¢¥o ¡ío¨öA/CI¡Æ¡© (AU¨ú¡ÀA¡×A¢®¡¤I AI¥ì¢¯)
; L112
LOAD      M02442	// IN-BUFF ALGN-FWD
OR        M18842	// T)IN-BUFF ALGN-FWD
LOAD      F00094
AND       M01910
OR LOAD
AND NOT   M00908	// IN-BUFF ALIGN Au/EAA©ª ¨úE¢Ò¡À
OUT       P0009A	// IN-BUFF ALGN-FWD
// ======================== AoAO¨¬I ¨ùO ¥ìe¨úi ¢¯O¢¥U ©ø¨£¡Æ¡Ì¡ÆA A¨ùA¨Ï ==========================
// 
// ¨¬?¡Æ©¡ : AUTO LOAD AI©öC¡¤I,  LOAD OK ©ö¨­¡Æi ALIGN ¢¯I¡¤a¡¤I ¨ùoA¢´
; L116
LOAD      M00201	// LF_AUTO RUN
AND       T2001	// IN-TRANS BUFF RIGHT     (L-LD)
AND NOT   P00014	// FRONT SAFETY SENSOR
OR        M18200	// ¢¯¨­AE ¨ùO¥ìe¨úi¢¯E
AND NOT   K00252	// LOADING ¡¾a ONLINE
AND NOT   M18100	// L_IN BUFFER VC ON
OUT       M18200	// ¢¯¨­AE ¨ùO¥ìe¨úi¢¯E
TON       T1190 200
; L118
LOAD      M00211	// RT_AUTO RUN
AND       T2000	// IN-TRANS     BUFF     LEFT     (R-LD)
AND NOT   P00014	// FRONT SAFETY SENSOR
OR        M18201	// ¢¯A¢¬¡ÍAE ¨ùO¥ìe¨úi¢¯E
AND NOT   K00252	// LOADING ¡¾a ONLINE
AND NOT   M18600	// R_IN BUFFER VC ON
OUT       M18201	// ¢¯A¢¬¡ÍAE ¨ùO¥ìe¨úi¢¯E
TON       T1191 200
// output comment: ¨ùo¥ì¢¯AoAOCuAA Aa¨¬n¢¯¢® AoAO¨¬I ¨¬o¨ù¨ú¨ù¡©¡Æ¢® 1¡Æ©ø¡¤I ¨¬?¡Æ©¡(2021.12)
; L120
LOAD      P00014	// FRONT SAFETY SENSOR
AND       T1190
AND       T2001	// IN-TRANS BUFF RIGHT     (L-LD)
AND       P0002A	// L_IN BUFF ROTATE     LD
AND NOT   K00252	// LOADING ¡¾a ONLINE
OUT       M18202	// ¢¯¨­AE ¨ùO©ø¨£¡Æ¡§
// output comment: ¡¾aA¢¬ AU¨ú¡ÀAU ¨ùO ¨¬uA¢ç ©ø¨£¡Æ¢®¢¥A¡ÆI ¡Æ¡§AoC¨ª¨ù¡© A©ª¡Æ©ª CI¢¥©ª¡ÆIA¡í AUTO LOAD EA ALIGN ¥ì¢¯AU CI¢¬e A©ª¡Æ©ªCI¡ÆO ¨ùoA¢´

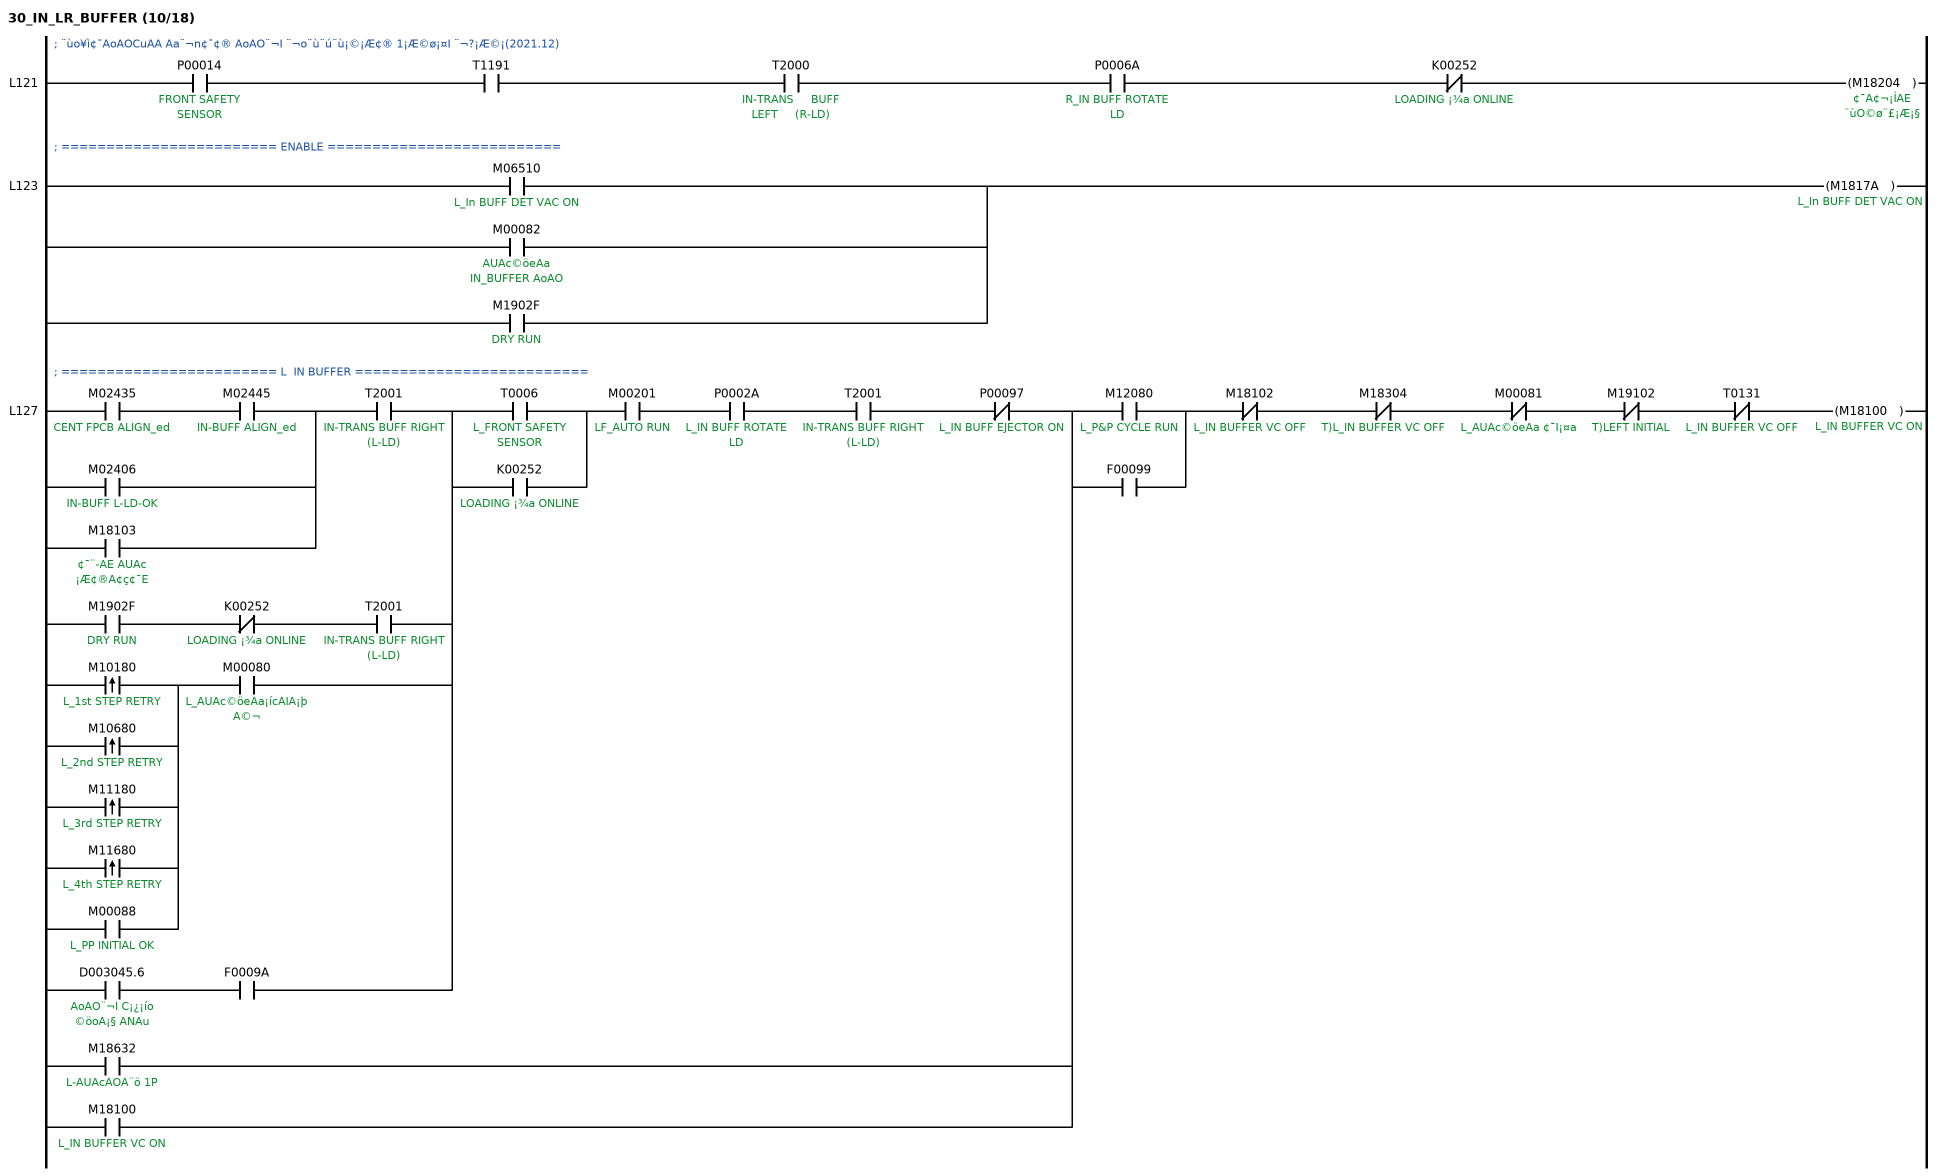
; L121
LOAD      P00014	// FRONT SAFETY SENSOR
AND       T1191
AND       T2000	// IN-TRANS     BUFF     LEFT     (R-LD)
AND       P0006A	// R_IN BUFF ROTATE      LD
AND NOT   K00252	// LOADING ¡¾a ONLINE
OUT       M18204	// ¢¯A¢¬¡ÍAE ¨ùO©ø¨£¡Æ¡§
// output comment: ¨ùo¥ì¢¯AoAOCuAA Aa¨¬n¢¯¢® AoAO¨¬I ¨¬o¨ù¨ú¨ù¡©¡Æ¢® 1¡Æ©ø¡¤I ¨¬?¡Æ©¡(2021.12)
// ======================== ENABLE ==========================
; L123
LOAD      M06510	// L_In BUFF DET VAC ON
OR        M00082	// AUAc©öeAa IN_BUFFER AoAO 
OR        M1902F	// DRY RUN
OUT       M1817A	// L_In BUFF DET VAC ON
// ======================== L  IN BUFFER ==========================
; L127
LOAD      M02435	// CENT FPCB ALIGN_ed
AND       M02445	// IN-BUFF ALIGN_ed
OR        M02406	// IN-BUFF L-LD-OK
OR        M18103	// ¢¯¨­AE AUAc ¡Æ¢®A¢ç¢¯E
AND       T2001	// IN-TRANS BUFF RIGHT     (L-LD)
LOAD      M1902F	// DRY RUN
AND NOT   K00252	// LOADING ¡¾a ONLINE
AND       T2001	// IN-TRANS BUFF RIGHT     (L-LD)
OR LOAD
LOADP     M10180	// L_1st STEP RETRY
ORP       M10680	// L_2nd STEP RETRY
ORP       M11180	// L_3rd STEP RETRY
ORP       M11680	// L_4th STEP RETRY
OR        M00088	// L_PP INITIAL OK
AND       M00080	// L_AUAc©öeAa¡ícAIA¡þA©¬
OR LOAD
LOAD      D003045.6	// AoAO¨¬I C¡¿¡ío ©öoA¡§ ANAu
AND       F0009A
OR LOAD
LOAD      T0006	// L_FRONT SAFETY SENSOR
OR        K00252	// LOADING ¡¾a ONLINE
AND LOAD
AND       M00201	// LF_AUTO RUN
AND       P0002A	// L_IN BUFF ROTATE     LD
AND       T2001	// IN-TRANS BUFF RIGHT     (L-LD)
AND NOT   P00097	// L_IN BUFF EJECTOR ON
OR        M18632	// L-AUAcAOA¨ö 1P
OR        M18100	// L_IN BUFFER VC ON
LOAD      M12080	// L_P&P CYCLE RUN
OR        F00099
AND LOAD
AND NOT   M18102	// L_IN BUFFER VC OFF
AND NOT   M18304	// T)L_IN BUFFER VC OFF
AND NOT   M00081	// L_AUAc©öeAa ¢¯I¡¤a
AND NOT   M19102	// T)LEFT INITIAL
AND NOT   T0131	// L_IN BUFFER VC OFF
OUT       M18100	// L_IN BUFFER VC ON

